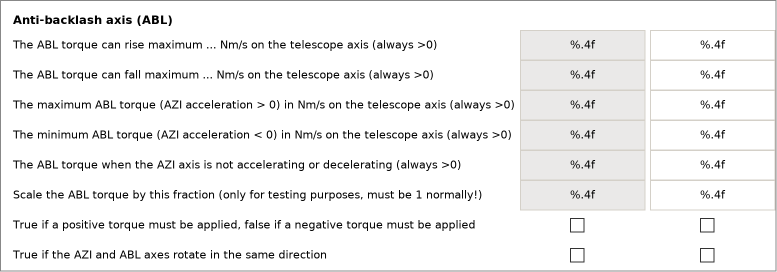
VISUALIZATION VISU_AxesConfig_Azimuth_3  // 777x272
VAR_IN_OUT
    active : AxesAzimuthConfig;
    editable : AxesAzimuthConfig;
END_VAR
    Label (10,5 205x30), "Anti-backlash axis (ABL)"
    Label (10,30 475x30), "The ABL torque can rise maximum ... Nm/s on the telescope axis (always >0)"
    Frame (520,30 255x30)
        shows VISU_ConfigLREAL4Entry(active := active.ablMaxTorqueRiseSpeed, editable := editable.ablMaxTorqueRiseSpeed)
    Label (10,60 475x30), "The ABL torque can fall maximum ... Nm/s on the telescope axis (always >0)"
    Label (10,90 505x30), "The maximum ABL torque (AZI acceleration > 0) in Nm/s on the telescope axis (always >0)"
    Label (10,120 500x30), "The minimum ABL torque (AZI acceleration < 0) in Nm/s on the telescope axis (always >0)"
    Label (10,150 500x30), "The ABL torque when the AZI axis is not accelerating or decelerating (always >0)"
    Label (10,180 500x30), "Scale the ABL torque by this fraction (only for testing purposes, must be 1 normally!)"
    Label (10,210 500x30), "True if a positive torque must be applied, false if a negative torque must be applied"
    Frame (520,210 255x30)
        shows VISU_ConfigBOOLEntry(active := active.ablPositiveTorque, editable := editable.ablPositiveTorque)
    Label (10,240 500x30), "True if the AZI and ABL axes rotate in the same direction"
    Frame (520,240 255x30)
        shows VISU_ConfigBOOLEntry(active := active.aziAndAblSameDirection, editable := editable.aziAndAblSameDirection)
    Frame (520,60 255x30)
        shows VISU_ConfigLREAL4Entry(active := active.ablMaxTorqueFallSpeed, editable := editable.ablMaxTorqueFallSpeed)
    Frame (520,90 255x30)
        shows VISU_ConfigLREAL4Entry(active := active.ablMaxTorque, editable := editable.ablMaxTorque)
    Frame (520,120 255x30)
        shows VISU_ConfigLREAL4Entry(active := active.ablMinTorque, editable := editable.ablMinTorque)
    Frame (520,150 255x30)
        shows VISU_ConfigLREAL4Entry(active := active.ablZeroAccTorque, editable := editable.ablZeroAccTorque)
    Frame (520,180 255x30)
        shows VISU_ConfigLREAL4Entry(active := active.ablTorqueOutputOverride, editable := editable.ablTorqueOutputOverride)
END_VISUALIZATION

// ---- MTCS/Axes/Visu/VISU_AxesConfig_Rotation_2.TcVIS
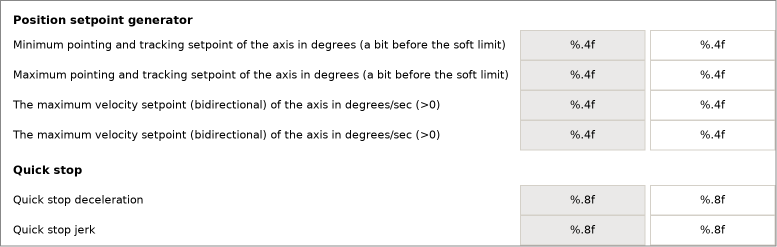
VISUALIZATION VISU_AxesConfig_Rotation_2  // 777x247
VAR_IN_OUT
    active : AxesRotationConfig;
    editable : AxesRotationConfig;
END_VAR
    Label (10,5 205x30), "Position setpoint generator"
    Label (10,30 495x30), "Minimum pointing and tracking setpoint of the axis in degrees (a bit before the soft limit)"
    Label (10,60 510x30), "Maximum pointing and tracking setpoint of the axis in degrees (a bit before the soft limit)"
    Label (10,90 475x30), "The maximum velocity setpoint (bidirectional) of the axis in degrees/sec (>0)"
    Label (10,120 475x30), "The maximum velocity setpoint (bidirectional) of the axis in degrees/sec (>0)"
    Frame (520,30 255x30)
        shows VISU_ConfigLREAL4Entry(active := active.minPositionSetpoint, editable := editable.minPositionSetpoint)
    Frame (520,60 255x30)
        shows VISU_ConfigLREAL4Entry(active := active.maxPositionSetpoint, editable := editable.maxPositionSetpoint)
    Frame (520,90 255x30)
        shows VISU_ConfigLREAL4Entry(active := active.maxVelocitySetpoint, editable := editable.maxVelocitySetpoint)
    Frame (520,120 255x30)
        shows VISU_ConfigLREAL4Entry(active := active.maxAccelerationSetpoint, editable := editable.maxAccelerationSetpoint)
    Label (10,155 205x30), "Quick stop"
    Frame (520,185 255x30)
        shows VISU_ConfigLREAL8Entry(active := active.quickStopDeceleration, editable := editable.quickStopDeceleration)
    Label (10,185 500x30), "Quick stop deceleration"
    Label (10,215 500x30), "Quick stop jerk"
    Frame (520,215 255x30)
        shows VISU_ConfigLREAL8Entry(active := active.quickStopJerk, editable := editable.quickStopJerk)
END_VISUALIZATION

// ---- MTCS/Axes/Visu/VISU_AxesConfig_Rotation_1.TcVIS
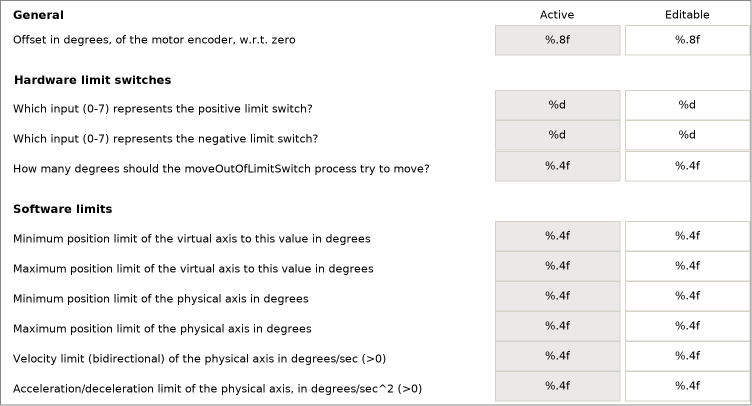
VISUALIZATION VISU_AxesConfig_Rotation_1  // 752x406
VAR_IN_OUT
    active : AxesRotationConfig;
    editable : AxesRotationConfig;
END_VAR
    Label (495,5 125x20), "Active"
    Label (625,5 125x20), "Editable"
    Label (10,25 360x30), "Offset in degrees, of the motor encoder, w.r.t. zero"
    Frame (495,25 255x30)
        shows VISU_ConfigLREAL8Entry(active := active.motorEncoderOffset, editable := editable.motorEncoderOffset)
    Label (10,94 475x30), "Which input (0-7) represents the positive limit switch?"
    Label (10,124 475x30), "Which input (0-7) represents the negative limit switch?"
    Label (10,154 475x30), "How many degrees should the moveOutOfLimitSwitch process try to move?"
    Label (11,65 150x30), "Hardware limit switches"
    Label (10,224 475x30), "Minimum position limit of the virtual axis to this value in degrees"
    Label (10,194 165x30), "Software limits"
    Label (10,254 475x30), "Maximum position limit of the virtual axis to this value in degrees"
    Label (10,284 475x30), "Minimum position limit of the physical axis in degrees"
    Label (10,314 475x30), "Maximum position limit of the physical axis in degrees"
    Label (10,344 475x30), "Velocity limit (bidirectional) of the physical axis in degrees/sec (>0)"
    Label (10,374 475x30), "Acceleration/deceleration limit of the physical axis, in degrees/sec^2 (>0)"
    Label (10,0 150x30), "General"
    Frame (495,90 255x30)
        shows VISU_ConfigSINTEntry(active := active.positiveLimitSwitchInput, editable := editable.positiveLimitSwitchInput)
    Frame (495,120 255x30)
        shows VISU_ConfigSINTEntry(active := active.negativeLimitSwitchInput, editable := editable.negativeLimitSwitchInput)
    Frame (495,151 255x30)
        shows VISU_ConfigLREAL4Entry(active := active.moveOutOfLimitSwitchDistance, editable := editable.moveOutOfLimitSwitchDistance)
    Frame (495,221 255x30)
        shows VISU_ConfigLREAL4Entry(active := active.minPositionLimitVirtualAxis, editable := editable.minPositionLimitVirtualAxis)
    Frame (495,251 255x30)
        shows VISU_ConfigLREAL4Entry(active := active.maxPositionLimitVirtualAxis, editable := editable.maxPositionLimitVirtualAxis)
    Frame (495,281 255x30)
        shows VISU_ConfigLREAL4Entry(active := active.minPositionLimitPhysicalAxis, editable := editable.minPositionLimitPhysicalAxis)
    Frame (495,311 255x30)
        shows VISU_ConfigLREAL4Entry(active := active.maxPositionLimitPhysicalAxis, editable := editable.maxPositionLimitPhysicalAxis)
    Frame (495,341 255x30)
        shows VISU_ConfigLREAL4Entry(active := active.velocityLimit, editable := editable.velocityLimit)
    Frame (495,371 255x30)
        shows VISU_ConfigLREAL4Entry(active := active.accelerationLimit, editable := editable.accelerationLimit)
END_VISUALIZATION

// ---- MTCS/Axes/Visu/VISU_AxesConfig_Elevation_2.TcVIS
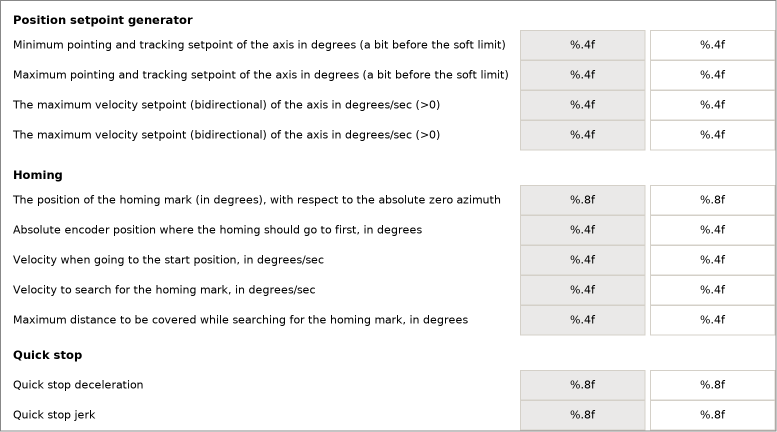
VISUALIZATION VISU_AxesConfig_Elevation_2  // 777x432
VAR_IN_OUT
    active : AxesElevationConfig;
    editable : AxesElevationConfig;
END_VAR
    Frame (520,185 255x30)
        shows VISU_ConfigLREAL8Entry(active := active.homingHomePosition, editable := editable.homingHomePosition)
    Label (10,185 500x30), "The position of the homing mark (in degrees), with respect to the absolute zero azimuth"
    Label (10,5 205x30), "Position setpoint generator"
    Label (10,30 490x30), "Minimum pointing and tracking setpoint of the axis in degrees (a bit before the soft limit)"
    Label (10,60 500x30), "Maximum pointing and tracking setpoint of the axis in degrees (a bit before the soft limit)"
    Label (10,90 475x30), "The maximum velocity setpoint (bidirectional) of the axis in degrees/sec (>0)"
    Label (10,120 475x30), "The maximum velocity setpoint (bidirectional) of the axis in degrees/sec (>0)"
    Label (10,160 205x30), "Homing"
    Label (10,215 475x30), "Absolute encoder position where the homing should go to first, in degrees"
    Label (10,245 475x30), "Velocity when going to the start position, in degrees/sec"
    Label (10,275 505x30), "Velocity to search for the homing mark, in degrees/sec"
    Label (10,305 500x30), "Maximum distance to be covered while searching for the homing mark, in degrees"
    Frame (520,30 255x30)
        shows VISU_ConfigLREAL4Entry(active := active.minPositionSetpoint, editable := editable.minPositionSetpoint)
    Frame (520,60 255x30)
        shows VISU_ConfigLREAL4Entry(active := active.maxPositionSetpoint, editable := editable.maxPositionSetpoint)
    Frame (520,90 255x30)
        shows VISU_ConfigLREAL4Entry(active := active.maxVelocitySetpoint, editable := editable.maxVelocitySetpoint)
    Frame (520,120 255x30)
        shows VISU_ConfigLREAL4Entry(active := active.maxAccelerationSetpoint, editable := editable.maxAccelerationSetpoint)
    Frame (520,215 255x30)
        shows VISU_ConfigLREAL4Entry(active := active.homingStartAbsEncPosition, editable := editable.homingStartAbsEncPosition)
    Frame (520,245 255x30)
        shows VISU_ConfigLREAL4Entry(active := active.homingGotoStartVelocity, editable := editable.homingGotoStartVelocity)
    Frame (520,275 255x30)
        shows VISU_ConfigLREAL4Entry(active := active.homingVelocity, editable := editable.homingVelocity)
    Frame (520,305 255x30)
        shows VISU_ConfigLREAL4Entry(active := active.homingRange, editable := editable.homingRange)
    Label (10,340 205x30), "Quick stop"
    Frame (520,370 255x30)
        shows VISU_ConfigLREAL8Entry(active := active.quickStopDeceleration, editable := editable.quickStopDeceleration)
    Label (10,370 500x30), "Quick stop deceleration"
    Label (10,400 500x30), "Quick stop jerk"
    Frame (520,400 255x30)
        shows VISU_ConfigLREAL8Entry(active := active.quickStopJerk, editable := editable.quickStopJerk)
END_VISUALIZATION

// ---- MTCS/Axes/Visu/VISU_AxesConfig_Elevation_1.TcVIS
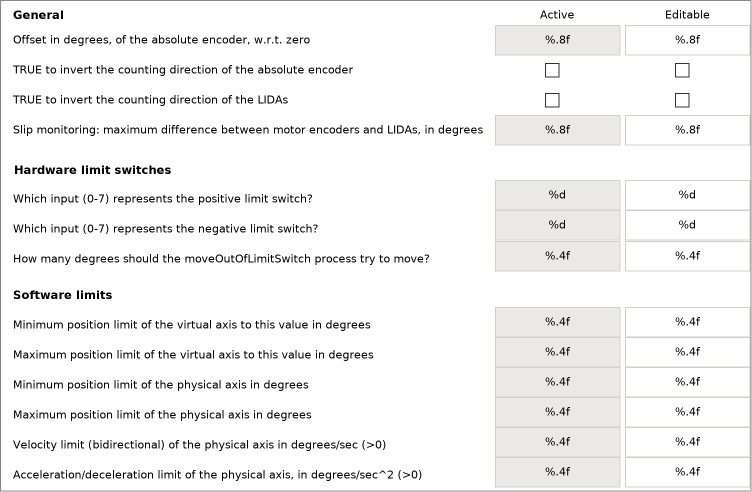
VISUALIZATION VISU_AxesConfig_Elevation_1  // 752x492
VAR_IN_OUT
    active : AxesElevationConfig;
    editable : AxesElevationConfig;
END_VAR
    Label (495,5 125x20), "Active"
    Label (625,5 125x20), "Editable"
    Label (10,25 360x30), "Offset in degrees, of the absolute encoder, w.r.t. zero"
    Frame (495,25 255x30)
        shows VISU_ConfigLREAL8Entry(active := active.absoluteEncoderOffset, editable := editable.absoluteEncoderOffset)
    Label (10,184 475x30), "Which input (0-7) represents the positive limit switch?"
    Label (10,214 475x30), "Which input (0-7) represents the negative limit switch?"
    Label (10,244 475x30), "How many degrees should the moveOutOfLimitSwitch process try to move?"
    Label (11,155 150x30), "Hardware limit switches"
    Label (10,310 475x30), "Minimum position limit of the virtual axis to this value in degrees"
    Label (10,280 165x30), "Software limits"
    Label (10,340 475x30), "Maximum position limit of the virtual axis to this value in degrees"
    Label (10,370 475x30), "Minimum position limit of the physical axis in degrees"
    Label (10,400 475x30), "Maximum position limit of the physical axis in degrees"
    Label (10,430 475x30), "Velocity limit (bidirectional) of the physical axis in degrees/sec (>0)"
    Label (10,460 475x30), "Acceleration/deceleration limit of the physical axis, in degrees/sec^2 (>0)"
    Label (10,115 480x30), "Slip monitoring: maximum difference between motor encoders and LIDAs, in degrees"
    Frame (495,115 255x30)
        shows VISU_ConfigLREAL8Entry(active := active.slipLimit, editable := editable.slipLimit)
    Label (10,0 150x30), "General"
    Frame (495,180 255x30)
        shows VISU_ConfigSINTEntry(active := active.positiveLimitSwitchInput, editable := editable.positiveLimitSwitchInput)
    Frame (495,210 255x30)
        shows VISU_ConfigSINTEntry(active := active.negativeLimitSwitchInput, editable := editable.negativeLimitSwitchInput)
    Frame (495,241 255x30)
        shows VISU_ConfigLREAL4Entry(active := active.moveOutOfLimitSwitchDistance, editable := editable.moveOutOfLimitSwitchDistance)
    Frame (495,307 255x30)
        shows VISU_ConfigLREAL4Entry(active := active.minPositionLimitVirtualAxis, editable := editable.minPositionLimitVirtualAxis)
    Frame (495,337 255x30)
        shows VISU_ConfigLREAL4Entry(active := active.maxPositionLimitVirtualAxis, editable := editable.maxPositionLimitVirtualAxis)
    Frame (495,367 255x30)
        shows VISU_ConfigLREAL4Entry(active := active.minPositionLimitPhysicalAxis, editable := editable.minPositionLimitPhysicalAxis)
    Frame (495,397 255x30)
        shows VISU_ConfigLREAL4Entry(active := active.maxPositionLimitPhysicalAxis, editable := editable.maxPositionLimitPhysicalAxis)
    Frame (495,427 255x30)
        shows VISU_ConfigLREAL4Entry(active := active.velocityLimit, editable := editable.velocityLimit)
    Frame (495,457 255x30)
        shows VISU_ConfigLREAL4Entry(active := active.accelerationLimit, editable := editable.accelerationLimit)
    Frame (495,55 255x30)
        shows VISU_ConfigBOOLEntry(active := active.absoluteEncoderInvert, editable := editable.absoluteEncoderInvert)
    Label (10,55 360x30), "TRUE to invert the counting direction of the absolute encoder"
    Frame (495,85 255x30)
        shows VISU_ConfigBOOLEntry(active := active.lidasInvert, editable := editable.lidasInvert)
    Label (10,85 360x30), "TRUE to invert the counting direction of the LIDAs"
END_VISUALIZATION

// ---- MTCS/Axes/Visu/VISU_AxesConfig_Azimuth_2.TcVIS
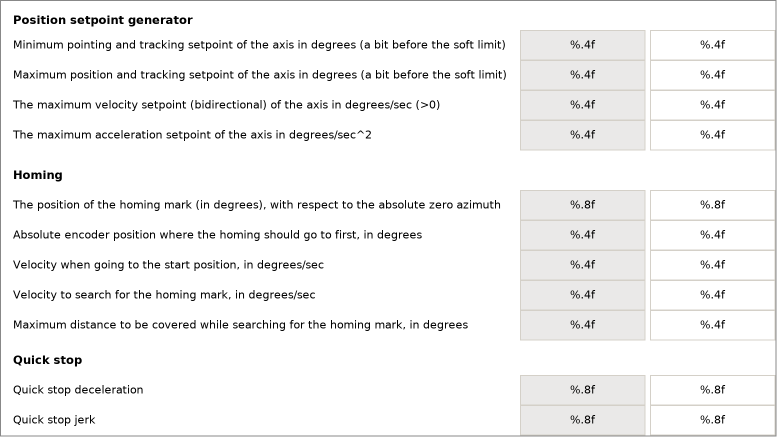
VISUALIZATION VISU_AxesConfig_Azimuth_2  // 777x437
VAR_IN_OUT
    active : AxesAzimuthConfig;
    editable : AxesAzimuthConfig;
END_VAR
    Frame (520,190 255x30)
        shows VISU_ConfigLREAL8Entry(active := active.homingHomePosition, editable := editable.homingHomePosition)
    Label (10,5 205x30), "Position setpoint generator"
    Label (10,30 500x30), "Minimum pointing and tracking setpoint of the axis in degrees (a bit before the soft limit)"
    Frame (520,30 255x30)
        shows VISU_ConfigLREAL4Entry(active := active.minPositionSetpoint, editable := editable.minPositionSetpoint)
    Label (10,60 500x30), "Maximum position and tracking setpoint of the axis in degrees (a bit before the soft limit)"
    Label (10,90 475x30), "The maximum velocity setpoint (bidirectional) of the axis in degrees/sec (>0)"
    Label (10,120 475x30), "The maximum acceleration setpoint of the axis in degrees/sec^2"
    Label (10,160 205x30), "Homing"
    Label (10,220 475x30), "Absolute encoder position where the homing should go to first, in degrees"
    Label (10,250 475x30), "Velocity when going to the start position, in degrees/sec"
    Label (10,280 505x30), "Velocity to search for the homing mark, in degrees/sec"
    Label (10,310 500x30), "Maximum distance to be covered while searching for the homing mark, in degrees"
    Frame (520,60 255x30)
        shows VISU_ConfigLREAL4Entry(active := active.maxPositionSetpoint, editable := editable.maxPositionSetpoint)
    Frame (520,90 255x30)
        shows VISU_ConfigLREAL4Entry(active := active.maxVelocitySetpoint, editable := editable.maxVelocitySetpoint)
    Frame (520,120 255x30)
        shows VISU_ConfigLREAL4Entry(active := active.maxAccelerationSetpoint, editable := editable.maxAccelerationSetpoint)
    Frame (520,220 255x30)
        shows VISU_ConfigLREAL4Entry(active := active.homingStartAbsEncPosition, editable := editable.homingStartAbsEncPosition)
    Frame (520,250 255x30)
        shows VISU_ConfigLREAL4Entry(active := active.homingGotoStartVelocity, editable := editable.homingGotoStartVelocity)
    Frame (520,280 255x30)
        shows VISU_ConfigLREAL4Entry(active := active.homingVelocity, editable := editable.homingVelocity)
    Frame (520,310 255x30)
        shows VISU_ConfigLREAL4Entry(active := active.homingRange, editable := editable.homingRange)
    Label (10,190 500x30), "The position of the homing mark (in degrees), with respect to the absolute zero azimuth"
    Label (10,345 205x30), "Quick stop"
    Frame (520,375 255x30)
        shows VISU_ConfigLREAL8Entry(active := active.quickStopDeceleration, editable := editable.quickStopDeceleration)
    Label (10,375 500x30), "Quick stop deceleration"
    Label (10,405 500x30), "Quick stop jerk"
    Frame (520,405 255x30)
        shows VISU_ConfigLREAL8Entry(active := active.quickStopJerk, editable := editable.quickStopJerk)
END_VISUALIZATION

// ---- MTCS/Axes/Visu/VISU_AxesConfig_FilterWheel.TcVIS
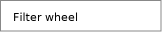
VISUALIZATION VISU_AxesConfig_FilterWheel  // 162x32
    Label (10,5 150x25), "Filter wheel"
END_VISUALIZATION

// ---- MTCS/Axes/Visu/VISU_AxesElevationAxis.TcVIS
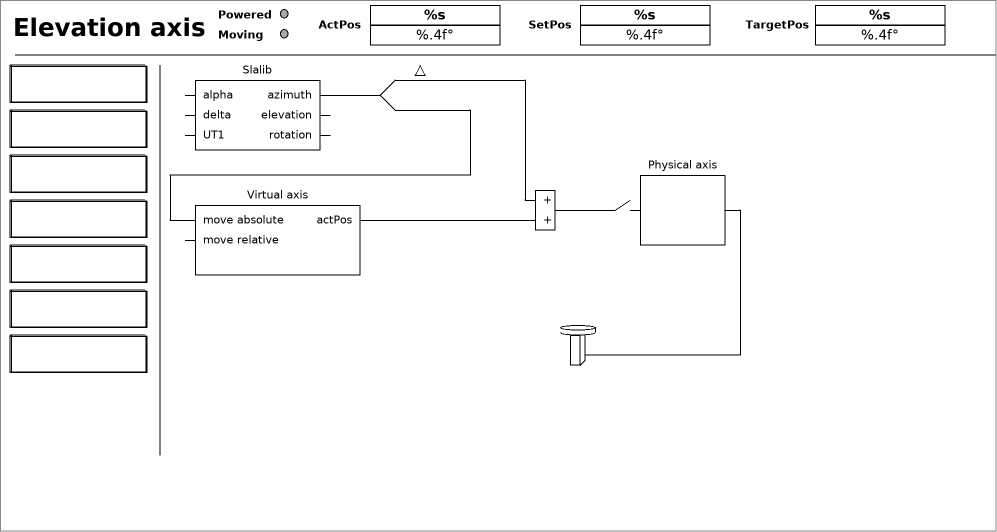
VISUALIZATION VISU_AxesElevationAxis  // 997x532
VAR_IN_OUT
	ref : AxesElevationAxis;
    ref_driveChannel : AX52XXDriveChannel;
    widget : AxesElevationAxisWidget;
END_VAR
    Rectangle (10,5 590x45), "Elevation axis"
    Frame (10,65 140x40)
        shows VISU_SubSubSystemButton(widget := widget.button_overview)
        OnMouseClick: FrameSelectionChange Selection=SelectedFrame=e720f99c-78fc-49d3-920d-5c22fdf0231f, GlobSel=AssignType=Directly, SelType=Locally
        OnMouseClick: execute { widget.activeTab := AxesElevationAxisTabs.OVERVIEW; }
    Frame (165,60 805x470)
        shows VISU_AxesElevationAxis_Overview(ref := ref, widget := widget)
        shows VISU_AxesElevationAxis_Processes(ref := ref, ref_driveChannel := ref_driveChannel, widget := widget)
        shows VISU_AX522DriveChannel(ref := ref_driveChannel, widget := widget.driveChannel)
        shows VISU_AngularAxis(axis := ref.parts.virtualAxis, widget := widget.virtualAxis)
        shows VISU_AngularAxis(axis := ref.parts.physicalAxis, widget := widget.physicalAxis)
        shows VISU_AxesElevationAxis_Lidas(ref := ref, widget := widget)
        shows VISU_AxesElevationAxis_AbsoluteEncoder(ref := ref, widget := widget)
        shows VISU_AxesAzimuthAxis_AbsoluteEncoder(ref := ref, widget := widget)
        p3523098516: ref
    Line (160,455) (160,65)
    Frame (10,155 140x40)
        shows VISU_SubSubSystemButton(widget := widget.button_driveChannel)
        OnMouseClick: FrameSelectionChange Selection=SelectedFrame=e720f99c-78fc-49d3-920d-5c22fdf0231f, Selection=2, GlobSel=AssignType=Directly, SelType=Locally
        OnMouseClick: execute { widget.activeTab := AxesElevationAxisTabs.DRIVE_CHANNEL; }
    Frame (10,200 140x40)
        shows VISU_SubSubSystemButton(widget := widget.button_virtualAxis)
        OnMouseClick: FrameSelectionChange Selection=SelectedFrame=e720f99c-78fc-49d3-920d-5c22fdf0231f, Selection=3, GlobSel=AssignType=Directly, SelType=Locally
        OnMouseClick: execute { widget.activeTab := AxesElevationAxisTabs.VIRTUAL_AXIS; }
    Frame (10,245 140x40)
        shows VISU_SubSubSystemButton(widget := widget.button_physicalAxis)
        OnMouseClick: FrameSelectionChange Selection=SelectedFrame=e720f99c-78fc-49d3-920d-5c22fdf0231f, Selection=4, GlobSel=AssignType=Directly, SelType=Locally
        OnMouseClick: execute { widget.activeTab := AxesElevationAxisTabs.PHYSICAL_AXIS; }
    Frame (10,290 140x40)
        shows VISU_SubSubSystemButton(widget := widget.button_lidas)
        OnMouseClick: FrameSelectionChange Selection=SelectedFrame=e720f99c-78fc-49d3-920d-5c22fdf0231f, Selection=5, GlobSel=AssignType=Directly, SelType=Locally
        OnMouseClick: execute { widget.activeTab := AxesElevationAxisTabs.LIDAS; }
    Frame (10,335 140x40)
        shows VISU_SubSubSystemButton(widget := widget.button_absoluteEncoder)
        OnMouseClick: FrameSelectionChange Selection=SelectedFrame=e720f99c-78fc-49d3-920d-5c22fdf0231f, Selection=6, GlobSel=AssignType=Directly, SelType=Locally
        OnMouseClick: execute { widget.activeTab := AxesElevationAxisTabs.ABSOLUTE_ENCODER; }
    Frame (10,110 140x40)
        shows VISU_SubSubSystemButton(widget := widget.button_processes)
        OnMouseClick: FrameSelectionChange Selection=SelectedFrame=e720f99c-78fc-49d3-920d-5c22fdf0231f, Selection=1, GlobSel=AssignType=Directly, SelType=Locally
        OnMouseClick: execute { widget.activeTab := AxesElevationAxisTabs.PROCESSES; }
    Line (995,55) (15,55)
    Label (310,0 60x50), "ActPos"
    Rectangle (370,5 130x20), "%s", text variable: widget.actPos.dmsString
    Rectangle (370,25 130x20), "%.4f°", text variable: ref.actPos.degrees.value
    Label (520,0 60x50), "SetPos"
    Rectangle (580,5 130x20), "%s", text variable: widget.setPos.dmsString
    Rectangle (580,25 130x20), "%.4f°", text variable: ref.setPos.degrees.value
    Label (740,0 75x50), "TargetPos"
    Rectangle (815,5 130x20), "%s", text variable: widget.targetPos.dmsString
    Rectangle (815,25 130x20), "%.4f°", text variable: ref.targetPos.degrees.value
    Label (215,5 65x20), "Powered"
    Frame (280,5 10x15)
        shows VISU_State_gray_green(state := ref.statuses.poweredStatus.enabled)
    Label (215,25 65x20), "Moving"
    Frame (280,25 10x15)
        shows VISU_State_gray_green(state := ref.parts.physicalAxis.axis_ref.Status.Moving)
END_VISUALIZATION

// ---- MTCS/Axes/Visu/VISU_AxesExternalSetpointGenerator.TcVIS
VISUALIZATION VISU_AxesExternalSetpointGenerator  // 2x2
END_VISUALIZATION

// ---- MTCS/Axes/Visu/VISU_AxesRotationAxis.TcVIS
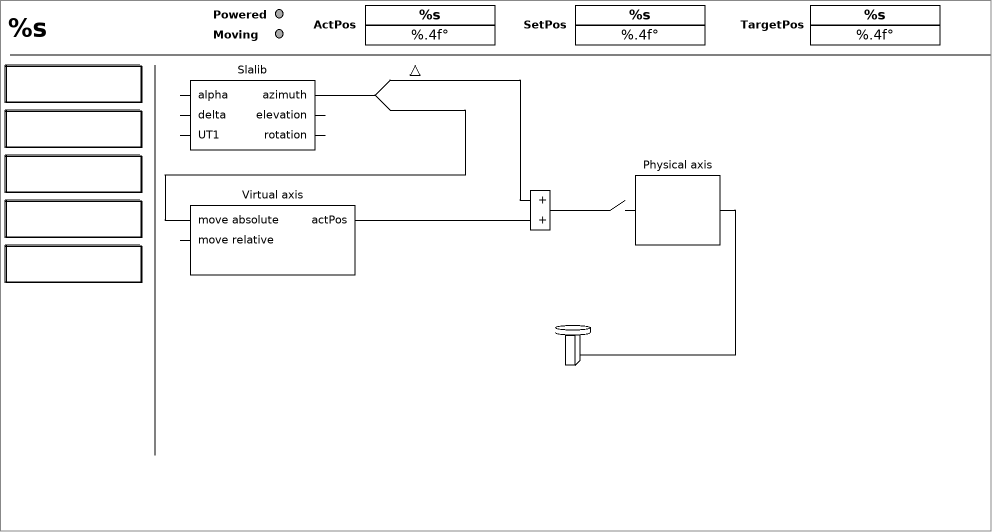
VISUALIZATION VISU_AxesRotationAxis  // 992x532
VAR_IN_OUT
	ref : AxesRotationAxis;
    ref_driveChannel : AX52XXDriveChannel;
    widget : AxesRotationAxisWidget;
END_VAR
    Frame (5,65 140x40)
        shows VISU_SubSubSystemButton(widget := widget.button_overview)
        OnMouseClick: FrameSelectionChange Selection=SelectedFrame=b6fa029b-3640-42a1-bfcc-db8ab31a5104, GlobSel=AssignType=Directly, SelType=Locally
        OnMouseClick: execute { widget.activeTab := AxesRotationAxisTabs.OVERVIEW; }
    Frame (160,60 805x470)
        shows VISU_AxesRotationAxis_Overview(ref := ref, widget := widget)
        shows VISU_AxesRotationAxis_Processes(ref := ref, ref_driveChannel := ref_driveChannel, widget := widget)
        shows VISU_AX522DriveChannel(ref := ref_driveChannel, widget := widget.driveChannel)
        shows VISU_AngularAxis(axis := ref.parts.virtualAxis, widget := widget.virtualAxis)
        shows VISU_AngularAxis(axis := ref.parts.physicalAxis, widget := widget.physicalAxis)
        shows VISU_AxesElevationAxis_AbsoluteEncoder(ref := ref, widget := widget)
        shows VISU_AxesAzimuthAxis_AbsoluteEncoder(ref := ref, widget := widget)
        shows VISU_AxesElevationAxis_Lidas(ref := ref, widget := widget)
        p3523098516: ref
    Line (155,455) (155,65)
    Frame (5,155 140x40)
        shows VISU_SubSubSystemButton(widget := widget.button_driveChannel)
        OnMouseClick: FrameSelectionChange Selection=SelectedFrame=b6fa029b-3640-42a1-bfcc-db8ab31a5104, Selection=2, GlobSel=AssignType=Directly, SelType=Locally
        OnMouseClick: execute { widget.activeTab := AxesRotationAxisTabs.DRIVE_CHANNEL; }
    Frame (5,200 140x40)
        shows VISU_SubSubSystemButton(widget := widget.button_virtualAxis)
        OnMouseClick: FrameSelectionChange Selection=SelectedFrame=b6fa029b-3640-42a1-bfcc-db8ab31a5104, Selection=3, GlobSel=AssignType=Directly, SelType=Locally
        OnMouseClick: execute { widget.activeTab := AxesRotationAxisTabs.VIRTUAL_AXIS; }
    Frame (5,245 140x40)
        shows VISU_SubSubSystemButton(widget := widget.button_physicalAxis)
        OnMouseClick: FrameSelectionChange Selection=SelectedFrame=b6fa029b-3640-42a1-bfcc-db8ab31a5104, Selection=4, GlobSel=AssignType=Directly, SelType=Locally
        OnMouseClick: execute { widget.activeTab := AxesRotationAxisTabs.PHYSICAL_AXIS; }
    Frame (5,110 140x40)
        shows VISU_SubSubSystemButton(widget := widget.button_processes)
        OnMouseClick: FrameSelectionChange Selection=SelectedFrame=b6fa029b-3640-42a1-bfcc-db8ab31a5104, Selection=1, GlobSel=AssignType=Directly, SelType=Locally
        OnMouseClick: execute { widget.activeTab := AxesRotationAxisTabs.PROCESSES; }
    Line (990,55) (10,55)
    Label (305,0 60x50), "ActPos"
    Rectangle (365,5 130x20), "%s", text variable: widget.actPos.dmsString
    Rectangle (365,25 130x20), "%.4f°", text variable: ref.actPos.degrees.value
    Label (515,0 60x50), "SetPos"
    Rectangle (575,5 130x20), "%s", text variable: widget.setPos.dmsString
    Rectangle (575,25 130x20), "%.4f°", text variable: ref.setPos.degrees.value
    Label (735,0 75x50), "TargetPos"
    Rectangle (810,5 130x20), "%s", text variable: widget.targetPos.dmsString
    Rectangle (810,25 130x20), "%.4f°", text variable: ref.targetPos.degrees.value
    Label (210,5 65x20), "Powered"
    Frame (275,5 10x15)
        shows VISU_State_gray_green(state := ref.statuses.poweredStatus.enabled)
    Label (210,25 65x20), "Moving"
    Frame (275,25 10x15)
        shows VISU_State_gray_green(state := ref.parts.physicalAxis.axis_ref.Status.Moving)
    Rectangle (5,5 200x46), "%s", text variable: widget.axisTitle
END_VISUALIZATION

// ---- MTCS/Axes/Visu/VISU_AxesManual.TcVIS
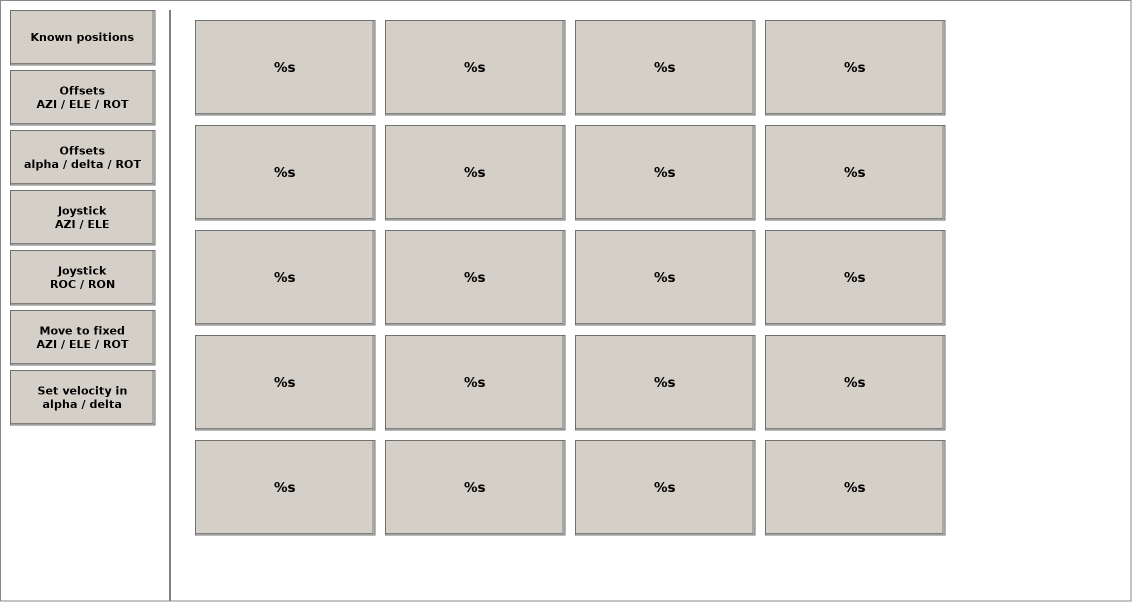
VISUALIZATION VISU_AxesManual  // 1132x602
VAR_IN_OUT
	ref : Axes;
    widget : AxesManualWidget;
END_VAR
    Button (10,10 145x55), "Known positions", pressed state: widget.activeTab = AxesManualTabs.TAB_POSITIONS
        OnMouseClick: execute { widget.activeTab := AxesManualTabs.TAB_POSITIONS; }
    Button (10,190 145x55), "Joystick AZI / ELE", pressed state: widget.activeTab = AxesManualTabs.TAB_JOYSTICK_AZIELE
        OnMouseClick: execute { widget.activeTab := AxesManualTabs.TAB_JOYSTICK_AZIELE; }
    Button (10,250 145x55), "Joystick ROC / RON", pressed state: widget.activeTab = AxesManualTabs.TAB_JOYSTICK_ROT
        OnMouseClick: execute { widget.activeTab := AxesManualTabs.TAB_JOYSTICK_ROT; }
    Button (10,70 145x55), "Offsets AZI / ELE / ROT", pressed state: widget.activeTab = AxesManualTabs.TAB_OFFSETS_AZIELE
        OnMouseClick: execute { widget.activeTab := AxesManualTabs.TAB_OFFSETS_AZIELE; }
    Button (10,310 145x55), "Move to fixed AZI / ELE / ROT", pressed state: widget.activeTab = AxesManualTabs.TAB_MOVEABSOLUTE
        OnMouseClick: execute { widget.activeTab := AxesManualTabs.TAB_MOVEABSOLUTE; }
    Button (10,370 145x55), "Set velocity in alpha / delta", pressed state: widget.activeTab = AxesManualTabs.TAB_MOVEVELOCITY
        OnMouseClick: execute { widget.activeTab := AxesManualTabs.TAB_MOVEVELOCITY; }
    Line (170,600) (170,10)
    Frame (180,10 950x590), frame switch variable: widget.activeTab
        shows VISU_AxesManual_Positions(ref := ref, widget := widget.positions)
        shows VISU_AxesManual_Joystick_AziEle(ref := ref, widget := widget.joystickAziEle)
        shows VISU_AxesManual_Joystick_Rot(ref := ref, widget := widget.joystickRot)
        shows VISU_AxesManual_Offsets_AziEleRot(ref := ref, widget := widget.offsets)
        shows VISU_AxesManual_Offsets_AlphaDeltaRot(ref := ref, widget := widget.offsets)
        shows VISU_AxesManual_MoveAbsolute(ref := ref, widget := widget.moveAbsolute)
        shows VISU_AxesManual_MoveVelocity(ref := ref, widget := widget.moveVelocity)
    Button (10,130 145x55), "Offsets alpha / delta / ROT", pressed state: widget.activeTab = AxesManualTabs.TAB_OFFSETS_ALPHADELTA
        OnMouseClick: execute { widget.activeTab := AxesManualTabs.TAB_OFFSETS_ALPHADELTA; }
END_VISUALIZATION

// ---- MTCS/Axes/Visu/VISU_AxesConfig.TcVIS
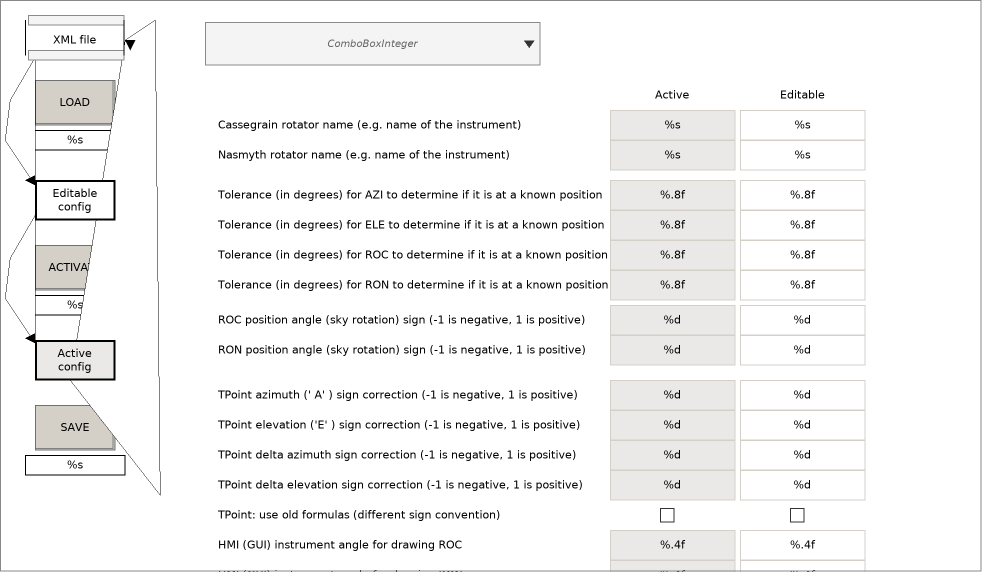
VISUALIZATION VISU_AxesConfig  // 982x572
VAR_IN_OUT
    editable : AxesConfig;
	active : AxesConfig;
    mgr : ConfigManager;
    mgrWidget : ConfigManagerWidget;
    axesWidget : AxesWidget;
END_VAR
    Frame (10,5 180x495)
        shows VISU_ConfigManager(mgr := mgr, widget := mgrWidget)
    ComboBoxInteger (205,22 335x43), variable: axesWidget.activeConfigTab, text list: 'AxesConfigTextList'
    Frame (205,85 775x485), frame switch variable: axesWidget.activeConfigTab
        shows VISU_AxesConfig_General(editable := editable, active := active)
        shows VISU_AxesConfig_KnownPositions(activePosition := axesWidget.activeConfigPosition, editable := editable.knownPositions, active := active.knownPositions)
        shows VISU_AxesConfig_Location(active := active.location, editable := editable.location)
        shows VISU_AxesConfig_LocalConditions(active := active.localConditions, editable := editable.localConditions)
        shows VISU_AxesConfig_Azimuth_1(active := active.azi, editable := editable.azi)
        shows VISU_AxesConfig_Azimuth_2(active := active.azi, editable := editable.azi)
        shows VISU_AxesConfig_Azimuth_3(active := active.azi, editable := editable.azi)
        shows VISU_AxesConfig_Elevation_1(active := active.ele, editable := editable.ele)
        shows VISU_AxesConfig_Elevation_2(active := active.ele, editable := editable.ele)
        shows VISU_AxesConfig_Rotation_1(active := active.roc, editable := editable.roc)
        shows VISU_AxesConfig_Rotation_2(active := active.roc, editable := editable.roc)
        shows VISU_AxesConfig_Rotation_1(active := active.ron, editable := editable.ron)
        shows VISU_AxesConfig_Rotation_2(active := active.ron, editable := editable.ron)
        shows VISU_AxesConfig_FilterWheel()
        shows VISU_MeasurementConfig(active := active.relativeHumidities.insideTube, editable := editable.relativeHumidities.insideTube)
        shows VISU_MeasurementConfig(active := active.dewpoints.topAir, editable := editable.dewpoints.topAir)
        shows VISU_MeasurementConfig(active := active.dewpoints.insideTube, editable := editable.dewpoints.insideTube)
        shows VISU_MeasurementConfig(active := active.accelerometers.tube.x, editable := editable.accelerometers.tube.x)
        shows VISU_MeasurementConfig(active := active.accelerometers.tube.y, editable := editable.accelerometers.tube.y)
        p1226617324: active.relativeHumidities.topAir
        p1437654724: editable.relativeHumidities.topAir
END_VISUALIZATION

// ---- MTCS/Axes/Visu/VISU_AxesAxes.TcVIS
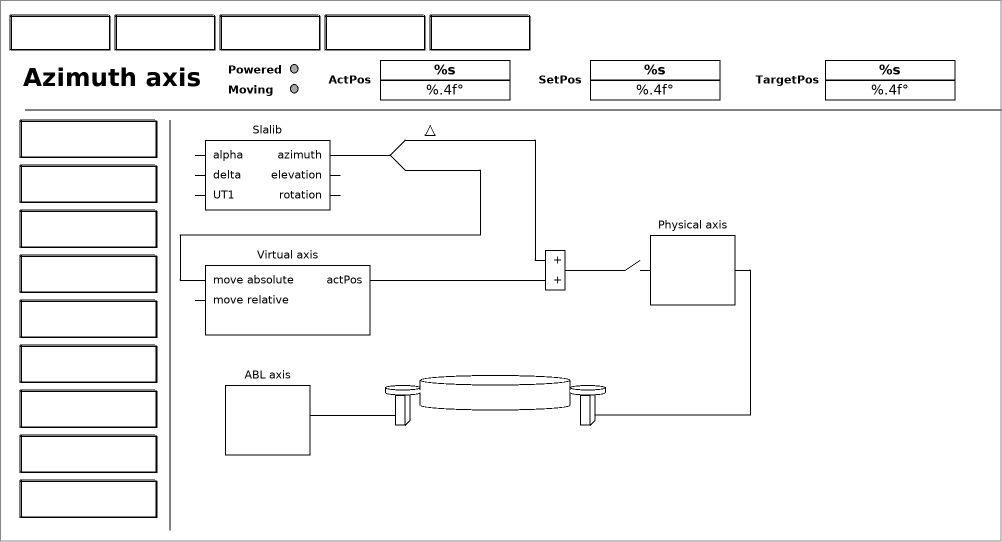
VISUALIZATION VISU_AxesAxes  // 1002x542
VAR_IN_OUT
    ref : Axes;
    widget : AxesAxesWidget;
END_VAR
    Frame (10,15 100x40)
        shows VISU_SubSubSystemButton(widget := widget.button_azi)
        OnMouseClick: FrameSelectionChange Selection=SelectedFrame=849b1b6c-774b-4476-bff7-38dbb17a175e, GlobSel=AssignType=Directly, SelType=Locally
        OnMouseClick: execute { widget.activeTab := AxesAxesTabs.AZI; }
    Frame (10,55 990x485)
        shows VISU_AxesAzimuthAxis(ref := ref.parts.azi, ref_aziDriveChannel := ref.parts.io.parts.aziDrive.parts.channelA, ref_ablDriveChannel := ref.parts.io.parts.ablDrive.parts.channelA, widget := widget.azi)
        shows VISU_AxesElevationAxis(ref := ref.parts.ele, ref_driveChannel := ref.parts.io.parts.eleDrive.parts.channelA, widget := widget.ele)
        shows VISU_AxesRotationAxis(ref := ref.parts.roc, ref_driveChannel := ref.parts.io.parts.aziDrive.parts.channelB, widget := widget.roc)
        shows VISU_AxesRotationAxis(ref := ref.parts.ron, ref_driveChannel := ref.parts.io.parts.ablDrive.parts.channelB, widget := widget.ron)
    Frame (115,15 100x40)
        shows VISU_SubSubSystemButton(widget := widget.button_ele)
        OnMouseClick: FrameSelectionChange Selection=SelectedFrame=849b1b6c-774b-4476-bff7-38dbb17a175e, Selection=1, GlobSel=AssignType=Directly, SelType=Locally
        OnMouseClick: execute { widget.activeTab := AxesAxesTabs.ELE; }
    Frame (220,15 100x40)
        shows VISU_SubSubSystemButton(widget := widget.button_roc)
        OnMouseClick: FrameSelectionChange Selection=SelectedFrame=849b1b6c-774b-4476-bff7-38dbb17a175e, Selection=2, GlobSel=AssignType=Directly, SelType=Locally
        OnMouseClick: execute { widget.activeTab := AxesAxesTabs.ROC; }
    Frame (325,15 100x40)
        shows VISU_SubSubSystemButton(widget := widget.button_ron)
        OnMouseClick: FrameSelectionChange Selection=SelectedFrame=849b1b6c-774b-4476-bff7-38dbb17a175e, Selection=3, GlobSel=AssignType=Directly, SelType=Locally
        OnMouseClick: execute { widget.activeTab := AxesAxesTabs.RON; }
    Frame (430,15 100x40)
        shows VISU_SubSubSystemButton(widget := widget.button_fw)
        OnMouseClick: FrameSelectionChange Selection=SelectedFrame=849b1b6c-774b-4476-bff7-38dbb17a175e, GlobSel=AssignType=Directly, SelType=Locally
        OnMouseClick: execute { widget.activeTab := AxesAxesTabs.FW; }
END_VISUALIZATION

// ---- MTCS/Axes/Visu/VISU_AxesAdvanced.TcVIS
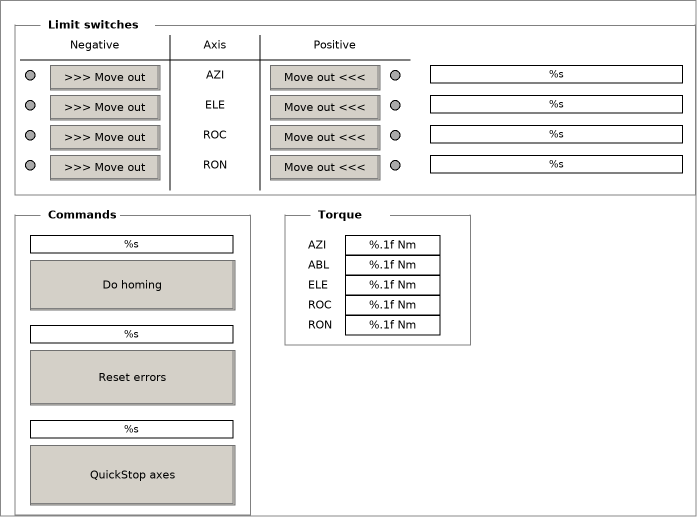
VISUALIZATION VISU_AxesAdvanced  // 697x517
VAR_IN_OUT
	ref : Axes;
    widget : AxesWidget;
END_VAR
    Polyline (120,215) (250,215) (250,515) (15,515) (15,215) (40,215)
    Polyline (155,25) (695,25) (695,195) (15,195) (15,25) (40,25)
    Label (45,15 100x20), "Limit switches"
    Label (170,60 90x30), "AZI"
    Frame (390,65 20x20)
        shows VISU_State_gray_red(state := ref.parts.azi.positiveLimitSwitchError)
    Line (260,190) (260,35)
    Line (170,190) (170,35)
    Label (260,30 150x30), "Positive"
    Label (20,30 150x30), "Negative"
    Line (410,60) (20,60)
    Label (170,30 90x30), "Axis"
    Button (270,65 110x25), "Move out <<<", input disabled if: ref.parts.azi.processes.moveOutOfLimitSwitch.statuses.enabledStatus.disabled
        OnMouseClick: execute { ref.parts.azi.processes.moveOutOfLimitSwitch.set.switch := LimitSwitches.POSITIVE_LIMIT_SWITCH; ref.parts.azi.processes.moveOutOfLimitSwitch.do_request := TRUE; }
    Frame (25,65 20x20)
        shows VISU_State_gray_red(state := ref.parts.azi.negativeLimitSwitchError)
    Button (50,65 110x25), ">>> Move out", input disabled if: ref.parts.azi.processes.moveOutOfLimitSwitch.statuses.enabledStatus.disabled
        OnMouseClick: execute { ref.parts.azi.processes.moveOutOfLimitSwitch.set.switch := LimitSwitches.NEGATIVE_LIMIT_SWITCH; ref.parts.azi.processes.moveOutOfLimitSwitch.do_request := TRUE; }
    Label (170,90 90x30), "ELE"
    Frame (390,95 20x20)
        shows VISU_State_gray_red(state := ref.parts.ele.positiveLimitSwitchError)
    Button (270,95 110x25), "Move out <<<", input disabled if: ref.parts.ele.processes.moveOutOfLimitSwitch.statuses.enabledStatus.disabled
        OnMouseClick: execute { ref.parts.ele.processes.moveOutOfLimitSwitch.set.switch := LimitSwitches.POSITIVE_LIMIT_SWITCH; ref.parts.ele.processes.moveOutOfLimitSwitch.do_request := TRUE; }
    Frame (25,95 20x20)
        shows VISU_State_gray_red(state := ref.parts.ele.negativeLimitSwitchError)
    Button (50,95 110x25), ">>> Move out", input disabled if: ref.parts.ele.processes.moveOutOfLimitSwitch.statuses.enabledStatus.disabled
        OnMouseClick: execute { ref.parts.ele.processes.moveOutOfLimitSwitch.set.switch := LimitSwitches.NEGATIVE_LIMIT_SWITCH; ref.parts.ele.processes.moveOutOfLimitSwitch.do_request := TRUE; }
    Label (170,120 90x30), "ROC"
    Frame (390,125 20x20)
        shows VISU_State_gray_red(state := ref.parts.roc.positiveLimitSwitchError)
    Button (270,125 110x25), "Move out <<<", input disabled if: ref.parts.roc.processes.moveOutOfLimitSwitch.statuses.enabledStatus.disabled
        OnMouseClick: execute { ref.parts.roc.processes.moveOutOfLimitSwitch.set.switch := LimitSwitches.POSITIVE_LIMIT_SWITCH; ref.parts.roc.processes.moveOutOfLimitSwitch.do_request := TRUE; }
    Frame (25,125 20x20)
        shows VISU_State_gray_red(state := ref.parts.roc.negativeLimitSwitchError)
    Button (50,125 110x25), ">>> Move out", input disabled if: ref.parts.roc.processes.moveOutOfLimitSwitch.statuses.enabledStatus.disabled
        OnMouseClick: execute { ref.parts.roc.processes.moveOutOfLimitSwitch.set.switch := LimitSwitches.NEGATIVE_LIMIT_SWITCH; ref.parts.roc.processes.moveOutOfLimitSwitch.do_request := TRUE; }
    Label (170,150 90x30), "RON"
    Frame (390,155 20x20)
        shows VISU_State_gray_red(state := ref.parts.ron.positiveLimitSwitchError)
    Button (270,155 110x25), "Move out <<<", input disabled if: ref.parts.ron.processes.moveOutOfLimitSwitch.statuses.enabledStatus.disabled
        OnMouseClick: execute { ref.parts.ron.processes.moveOutOfLimitSwitch.set.switch := LimitSwitches.POSITIVE_LIMIT_SWITCH; ref.parts.ron.processes.moveOutOfLimitSwitch.do_request := TRUE; }
    Frame (25,155 20x20)
        shows VISU_State_gray_red(state := ref.parts.ron.negativeLimitSwitchError)
    Button (50,155 110x25), ">>> Move out", input disabled if: ref.parts.ron.processes.moveOutOfLimitSwitch.statuses.enabledStatus.disabled
        OnMouseClick: execute { ref.parts.ron.processes.moveOutOfLimitSwitch.set.switch := LimitSwitches.NEGATIVE_LIMIT_SWITCH; ref.parts.ron.processes.moveOutOfLimitSwitch.do_request := TRUE; }
    Frame (430,65 255x20)
        shows VISU_StatusWidget(widget := widget.axes.azi.processes_moveOutOfLimitSwitchStatus)
    Frame (430,95 255x20)
        shows VISU_StatusWidget(widget := widget.axes.ele.processes_moveOutOfLimitSwitchStatus)
    Frame (430,125 255x20)
        shows VISU_StatusWidget(widget := widget.axes.roc.processes_moveOutOfLimitSwitchStatus)
    Frame (430,155 255x20)
        shows VISU_StatusWidget(widget := widget.axes.ron.processes_moveOutOfLimitSwitchStatus)
    Button (30,260 205x50), "Do homing", input disabled if: ref.processes.doHoming.statuses.enabledStatus.disabled
        OnMouseClick: execute { ref.processes.doHoming.do_request := TRUE; }
    Label (45,205 85x20), "Commands"
    Button (30,350 205x55), "Reset errors", input disabled if: ref.processes.reset.statuses.enabledStatus.disabled
        OnMouseClick: execute { ref.processes.reset.do_request := TRUE; }
    Frame (30,325 205x20)
        shows VISU_StatusWidget(widget := widget.processes_resetStatus)
        p4168582468: ref.processes.reset.actualStatus
    Frame (30,235 205x20)
        shows VISU_StatusWidget(widget := widget.processes_doHomingStatus)
        p4168582468: ref.processes.doHoming.actualStatus
    Button (30,445 205x60), "QuickStop axes", input disabled if: ref.processes.quickStop.statuses.enabledStatus.disabled
        OnMouseClick: execute { ref.processes.quickStop.do_request := TRUE; }
    Frame (30,420 205x20)
        shows VISU_StatusWidget(widget := widget.processes_quickStopStatus)
        p4168582468: ref.processes.quickStop.actualStatus
    Label (305,235 40x20), "AZI"
    Rectangle (345,235 95x20), "%.1f Nm", text variable: ref.parts.azi.actTorqueAzi.newtonmeter.value
    Label (305,255 40x20), "ABL"
    Rectangle (345,255 95x20), "%.1f Nm", text variable: ref.parts.azi.actTorqueAbl.newtonmeter.value
    Label (305,275 40x20), "ELE"
    Rectangle (345,275 95x20), "%.1f Nm", text variable: ref.parts.ele.actTorque.newtonmeter.value
    Label (305,295 40x20), "ROC"
    Rectangle (345,295 95x20), "%.1f Nm", text variable: ref.parts.roc.actTorque.newtonmeter.value
    Label (305,315 40x20), "RON"
    Rectangle (345,315 95x20), "%.1f Nm", text variable: ref.parts.ron.actTorque.newtonmeter.value
    Polyline (390,215) (470,215) (470,345) (285,345) (285,215) (310,215)
    Label (315,205 60x20), "Torque"
END_VISUALIZATION

// ---- MTCS/Axes/Visu/VISU_AxesPointingModelConfig_part1.TcVIS
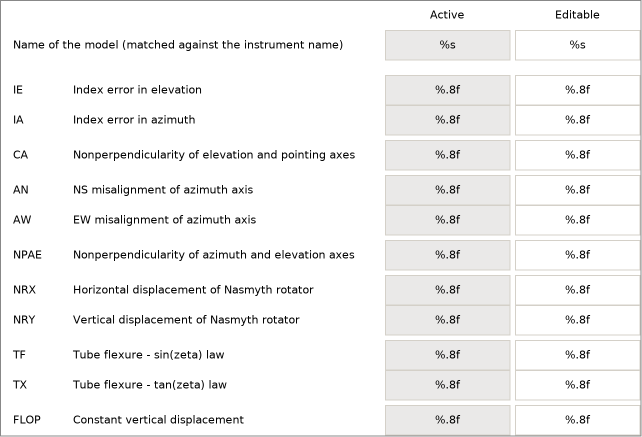
VISUALIZATION VISU_AxesPointingModelConfig_part1  // 642x437
VAR_IN_OUT
    active : AxesPointingModelConfig;
    editable : AxesPointingModelConfig;
END_VAR
    Label (385,5 125x20), "Active"
    Label (515,5 125x20), "Editable"
    Label (10,75 30x30), "IE"
    Frame (385,75 255x30)
        shows VISU_ConfigLREAL8Entry(active := active.IE, editable := editable.IE)
    Label (70,75 315x30), "Index error in elevation"
    Label (10,105 30x30), "IA"
    Frame (385,105 255x30)
        shows VISU_ConfigLREAL8Entry(active := active.IA, editable := editable.IA)
    Label (70,105 315x30), "Index error in azimuth"
    Label (10,140 30x30), "CA"
    Frame (385,140 255x30)
        shows VISU_ConfigLREAL8Entry(active := active.CA, editable := editable.CA)
    Label (70,140 315x30), "Nonperpendicularity of elevation and pointing axes"
    Label (10,175 30x30), "AN"
    Frame (385,175 255x30)
        shows VISU_ConfigLREAL8Entry(active := active.AN, editable := editable.AN)
    Label (70,175 315x30), "NS misalignment of azimuth axis"
    Frame (385,205 255x30)
        shows VISU_ConfigLREAL8Entry(active := active.AW, editable := editable.AW)
    Label (10,205 60x30), "AW"
    Label (70,205 315x30), "EW misalignment of azimuth axis"
    Frame (385,240 255x30)
        shows VISU_ConfigLREAL8Entry(active := active.NPAE, editable := editable.NPAE)
    Label (10,240 60x30), "NPAE"
    Label (70,240 315x30), "Nonperpendicularity of azimuth and elevation axes"
    Frame (385,275 255x30)
        shows VISU_ConfigLREAL8Entry(active := active.NRX, editable := editable.NRX)
    Label (10,275 60x30), "NRX"
    Label (70,275 315x30), "Horizontal displacement of Nasmyth rotator"
    Frame (385,305 255x30)
        shows VISU_ConfigLREAL8Entry(active := active.NRY, editable := editable.NRY)
    Label (10,305 60x30), "NRY"
    Label (70,305 315x30), "Vertical displacement of Nasmyth rotator"
    Frame (385,340 255x30)
        shows VISU_ConfigLREAL8Entry(active := active.TF, editable := editable.TF)
    Label (10,340 60x30), "TF"
    Label (70,340 315x30), "Tube flexure - sin(zeta) law"
    Frame (385,370 255x30)
        shows VISU_ConfigLREAL8Entry(active := active.TX, editable := editable.TX)
    Label (10,370 60x30), "TX"
    Label (70,370 315x30), "Tube flexure - tan(zeta) law"
    Frame (385,30 255x30)
        shows VISU_ConfigStringEntry(active := active.name, editable := editable.name)
    Label (10,30 370x30), "Name of the model (matched against the instrument name)"
    Frame (385,405 255x30)
        shows VISU_ConfigLREAL8Entry(active := active.FLOP, editable := editable.FLOP)
    Label (10,405 60x30), "FLOP"
    Label (70,405 315x30), "Constant vertical displacement"
END_VISUALIZATION

// ---- MTCS/Axes/Visu/VISU_AxesPointingModelConfig_part2.TcVIS
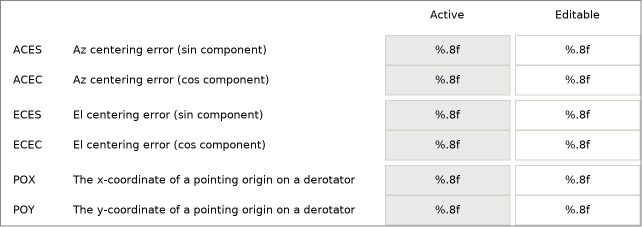
VISUALIZATION VISU_AxesPointingModelConfig_part2  // 642x227
VAR_IN_OUT
    active : AxesPointingModelConfig;
    editable : AxesPointingModelConfig;
END_VAR
    Label (385,5 125x20), "Active"
    Label (515,5 125x20), "Editable"
    Label (10,35 50x30), "ACES"
    Frame (385,35 255x30)
        shows VISU_ConfigLREAL8Entry(active := active.ACES, editable := editable.ACES)
    Label (70,35 315x30), "Az centering error (sin component)"
    Label (10,65 50x30), "ACEC"
    Frame (385,65 255x30)
        shows VISU_ConfigLREAL8Entry(active := active.ACEC, editable := editable.ACEC)
    Label (70,65 315x30), "Az centering error (cos component)"
    Label (10,100 50x30), "ECES"
    Frame (385,100 255x30)
        shows VISU_ConfigLREAL8Entry(active := active.ECES, editable := editable.ECES)
    Label (70,100 315x30), "El centering error (sin component)"
    Label (10,130 50x30), "ECEC"
    Frame (385,130 255x30)
        shows VISU_ConfigLREAL8Entry(active := active.ECEC, editable := editable.ECEC)
    Label (70,130 315x30), "El centering error (cos component)"
    Label (10,165 50x30), "POX"
    Frame (385,165 255x30)
        shows VISU_ConfigLREAL8Entry(active := active.POX, editable := editable.POX)
    Label (70,165 315x30), "The x-coordinate of a pointing origin on a derotator"
    Label (10,195 50x30), "POY"
    Frame (385,195 255x30)
        shows VISU_ConfigLREAL8Entry(active := active.POY, editable := editable.POY)
    Label (70,195 315x30), "The y-coordinate of a pointing origin on a derotator"
END_VISUALIZATION

// ---- MTCS/Axes/Visu/VISU_AxesPointingModelSetup.TcVIS
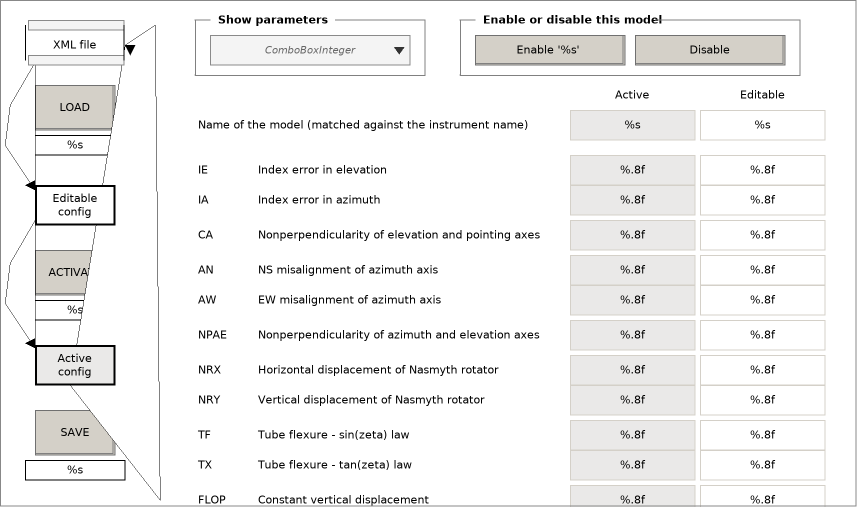
VISUALIZATION VISU_AxesPointingModelSetup  // 857x507
VAR_IN_OUT
    ref : AxesPointingModelSetup;
    widget : AxesPointingModelSetupWidget;
END_VAR
    Polyline (210,20) (195,20) (195,75) (425,75) (425,20) (335,20)
    Frame (10,10 180x495)
        shows VISU_ConfigManager(mgr := ref.parts.configManager, widget := widget.configManager)
    Frame (185,80 670x420), frame switch variable: widget.part
        shows VISU_AxesPointingModelConfig_part1(active := ref.config, editable := ref.editableConfig)
        shows VISU_AxesPointingModelConfig_part2(active := ref.config, editable := ref.editableConfig)
        shows VISU_MeasurementConfig(active := active.temperatures.m2Electronics, editable := editable.temperatures.m2Electronics)
        shows VISU_MeasurementConfig(active := active.temperatures.topTube, editable := editable.temperatures.topTube)
        shows VISU_MeasurementConfig(active := active.temperatures.centreTube, editable := editable.temperatures.centreTube)
        shows VISU_MeasurementConfig(active := active.temperatures.fork, editable := editable.temperatures.fork)
        shows VISU_MeasurementConfig(active := active.temperatures.nasmythAir, editable := editable.temperatures.nasmythAir)
        shows VISU_MeasurementConfig(active := active.temperatures.rem, editable := editable.temperatures.rem)
        shows VISU_MeasurementConfig(active := active.temperatures.rpm, editable := editable.temperatures.rpm)
        shows VISU_MeasurementConfig(active := active.temperatures.hermesTelescopeAdapter, editable := editable.temperatures.hermesTelescopeAdapter)
        shows VISU_MeasurementConfig(active := active.temperatures.topAir, editable := editable.temperatures.topAir)
        shows VISU_MeasurementConfig(active := active.temperatures.insideTube, editable := editable.temperatures.insideTube)
        shows VISU_MeasurementConfig(active := active.relativeHumidities.topAir, editable := editable.relativeHumidities.topAir)
        shows VISU_MeasurementConfig(active := active.relativeHumidities.insideTube, editable := editable.relativeHumidities.insideTube)
        shows VISU_MeasurementConfig(active := active.dewpoints.topAir, editable := editable.dewpoints.topAir)
        shows VISU_MeasurementConfig(active := active.dewpoints.insideTube, editable := editable.dewpoints.insideTube)
        shows VISU_MeasurementConfig(active := active.accelerometers.tube.x, editable := editable.accelerometers.tube.x)
        shows VISU_MeasurementConfig(active := active.accelerometers.tube.y, editable := editable.accelerometers.tube.y)
        shows VISU_AxesConfig_LocalConditions(active := active.localConditions, editable := editable.localConditions)
    ComboBoxInteger (210,35 200x30), variable: widget.part, text list: 'AxesPointingModelSetupPartsTextList'
    Label (480,10 180x20), "Enable or disable this model"
    Polyline (475,20) (460,20) (460,75) (800,75) (800,20) (655,20)
    Button (475,35 150x30), "Enable '%s'", text variable: ref.config.name, input disabled if: widget.enableButtonDisabled
        OnMouseClick: execute { widget.enableButtonPressed := TRUE; }
    Button (635,35 150x30), "Disable", input disabled if: widget.disableButtonDisabled
        OnMouseClick: execute { widget.disableButtonPressed := TRUE; }
    Label (215,10 125x20), "Show parameters"
END_VISUALIZATION

// ---- MTCS/Axes/Visu/VISU_AxesConfig_General.TcVIS
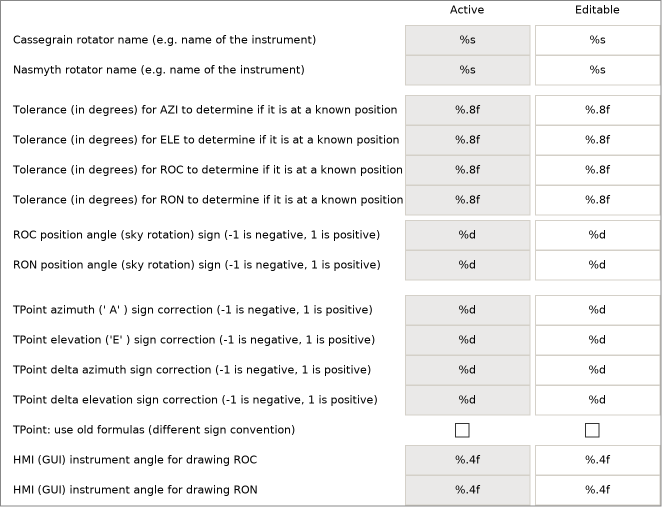
VISUALIZATION VISU_AxesConfig_General  // 662x507
VAR_IN_OUT
    editable : AxesConfig;
	active : AxesConfig;
END_VAR
    Frame (405,25 255x30)
        shows VISU_ConfigStringEntry(active := active.cassegrainRotatorName, editable := editable.cassegrainRotatorName)
    Label (405,0 125x20), "Active"
    Label (535,0 125x20), "Editable"
    Label (10,25 370x30), "Cassegrain rotator name (e.g. name of the instrument)"
    Frame (405,55 255x30)
        shows VISU_ConfigStringEntry(active := active.nasmythRotatorName, editable := editable.nasmythRotatorName)
    Label (10,55 370x30), "Nasmyth rotator name (e.g. name of the instrument)"
    Frame (405,95 255x30)
        shows VISU_ConfigLREAL8Entry(active := active.knownPositionToleranceAzi, editable := editable.knownPositionToleranceAzi)
    Label (10,95 395x30), "Tolerance (in degrees) for AZI to determine if it is at a known position"
    Label (10,125 395x30), "Tolerance (in degrees) for ELE to determine if it is at a known position"
    Frame (405,125 255x30)
        shows VISU_ConfigLREAL8Entry(active := active.knownPositionToleranceEle, editable := editable.knownPositionToleranceEle)
    Label (10,155 395x30), "Tolerance (in degrees) for ROC to determine if it is at a known position"
    Frame (405,155 255x30)
        shows VISU_ConfigLREAL8Entry(active := active.knownPositionToleranceRoc, editable := editable.knownPositionToleranceRoc)
    Label (10,185 395x30), "Tolerance (in degrees) for RON to determine if it is at a known position"
    Frame (405,185 255x30)
        shows VISU_ConfigLREAL8Entry(active := active.knownPositionToleranceRon, editable := editable.knownPositionToleranceRon)
    Frame (405,295 255x30)
        shows VISU_ConfigINTEntry(active := active.tpointAziSign, editable := editable.tpointAziSign)
    Label (10,295 395x30), "TPoint azimuth (' A' ) sign correction (-1 is negative, 1 is positive)"
    Frame (405,325 255x30)
        shows VISU_ConfigINTEntry(active := active.tpointEleSign, editable := editable.tpointEleSign)
    Label (10,325 395x30), "TPoint elevation ('E' ) sign correction (-1 is negative, 1 is positive)"
    Frame (405,355 255x30)
        shows VISU_ConfigINTEntry(active := active.tpointDeltaAziSign, editable := editable.tpointDeltaAziSign)
    Label (10,355 395x30), "TPoint delta azimuth sign correction (-1 is negative, 1 is positive)"
    Frame (405,385 255x30)
        shows VISU_ConfigINTEntry(active := active.tpointDeltaEleSign, editable := editable.tpointDeltaEleSign)
    Label (10,385 395x30), "TPoint delta elevation sign correction (-1 is negative, 1 is positive)"
    Label (10,415 395x30), "TPoint: use old formulas (different sign convention)"
    Frame (405,415 255x30)
        shows VISU_ConfigBOOLEntry(active := active.tpointOldFormulas, editable := editable.tpointOldFormulas)
    Frame (405,220 255x30)
        shows VISU_ConfigINTEntry(active := active.rocPositionAngleSign, editable := editable.rocPositionAngleSign)
    Label (10,220 395x30), "ROC position angle (sky rotation) sign (-1 is negative, 1 is positive)"
    Frame (405,250 255x30)
        shows VISU_ConfigINTEntry(active := active.ronPositionAngleSign, editable := editable.ronPositionAngleSign)
    Label (10,250 395x30), "RON position angle (sky rotation) sign (-1 is negative, 1 is positive)"
    Frame (405,445 255x30)
        shows VISU_ConfigLREAL4Entry(active := active.rocGuiAngle, editable := editable.rocGuiAngle)
    Label (10,445 395x30), "HMI (GUI) instrument angle for drawing ROC"
    Frame (405,475 255x30)
        shows VISU_ConfigLREAL4Entry(active := active.ronGuiAngle, editable := editable.ronGuiAngle)
    Label (10,475 395x30), "HMI (GUI) instrument angle for drawing RON"
END_VISUALIZATION

// ---- MTCS/Axes/Visu/VISU_AxesConfig_Location.TcVIS
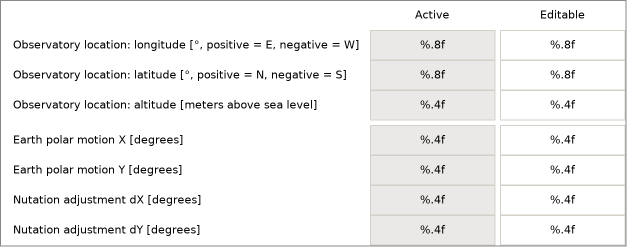
VISUALIZATION VISU_AxesConfig_Location  // 627x247
VAR_IN_OUT
    active : AxesLocationConfig;
    editable : AxesLocationConfig;
END_VAR
    Label (370,5 125x20), "Active"
    Label (500,5 125x20), "Editable"
    Label (10,30 360x30), "Observatory location: longitude [°, positive = E, negative = W]"
    Frame (370,30 255x30)
        shows VISU_ConfigLREAL8Entry(active := active.longitude, editable := editable.longitude)
    Frame (370,60 255x30)
        shows VISU_ConfigLREAL8Entry(active := active.latitude, editable := editable.latitude)
    Label (10,60 360x30), "Observatory location: latitude [°, positive = N, negative = S]"
    Label (10,90 360x30), "Observatory location: altitude [meters above sea level]"
    Frame (370,90 255x30)
        shows VISU_ConfigREAL4Entry(active := active.height, editable := editable.height)
    Label (10,125 360x30), "Earth polar motion X [degrees]"
    Frame (370,125 255x30)
        shows VISU_ConfigREAL4Entry(active := active.polarMotionX, editable := editable.polarMotionX)
    Label (10,155 360x30), "Earth polar motion Y [degrees]"
    Frame (370,155 255x30)
        shows VISU_ConfigREAL4Entry(active := active.polarMotionY, editable := editable.polarMotionY)
    Frame (370,185 255x30)
        shows VISU_ConfigREAL4Entry(active := active.nutationDx, editable := editable.nutationDx)
    Label (10,185 360x30), "Nutation adjustment dX [degrees]"
    Label (10,215 360x30), "Nutation adjustment dY [degrees]"
    Frame (370,215 255x30)
        shows VISU_ConfigREAL4Entry(active := active.nutationDy, editable := editable.nutationDy)
END_VISUALIZATION

// ---- MTCS/Axes/Visu/VISU_AxesConfig_LocalConditions.TcVIS
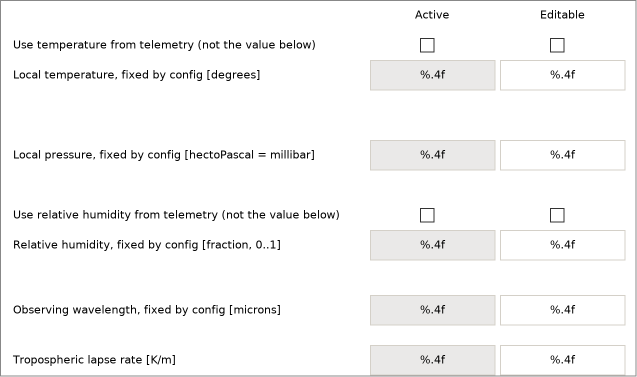
VISUALIZATION VISU_AxesConfig_LocalConditions  // 637x377
VAR_IN_OUT
    active : AxesLocalConditionsConfig;
    editable : AxesLocalConditionsConfig;
END_VAR
    Label (370,5 125x20), "Active"
    Label (500,5 125x20), "Editable"
    Label (10,30 360x30), "Use temperature from telemetry (not the value below)"
    Frame (370,30 265x30)
        shows VISU_ConfigBOOLEntry(active := active.useTemperatureFromSensors, editable := editable.useTemperatureFromSensors)
    Label (10,60 360x30), "Local temperature, fixed by config [degrees]"
    Frame (370,60 255x30)
        shows VISU_ConfigREAL4Entry(active := active.configuredTemperature, editable := editable.configuredTemperature)
    Label (10,140 360x30), "Local pressure, fixed by config [hectoPascal = millibar]"
    Frame (370,140 255x30)
        shows VISU_ConfigREAL4Entry(active := active.configuredPressure, editable := editable.configuredPressure)
    Label (10,230 360x30), "Relative humidity, fixed by config [fraction, 0..1]"
    Label (10,200 360x30), "Use relative humidity from telemetry (not the value below)"
    Frame (370,200 265x30)
        shows VISU_ConfigBOOLEntry(active := active.useRelativeHumidityFromSensors, editable := editable.useRelativeHumidityFromSensors)
    Frame (370,230 255x30)
        shows VISU_ConfigREAL4Entry(active := active.configuredRelativeHumidity, editable := editable.configuredRelativeHumidity)
    Label (10,295 360x30), "Observing wavelength, fixed by config [microns]"
    Frame (370,295 255x30)
        shows VISU_ConfigREAL4Entry(active := active.configuredObservingWavelength, editable := editable.configuredObservingWavelength)
    Label (10,345 360x30), "Tropospheric lapse rate [K/m]"
    Frame (370,345 255x30)
        shows VISU_ConfigREAL4Entry(active := active.troposphericLapseRate, editable := editable.troposphericLapseRate)
END_VISUALIZATION

// ---- MTCS/Axes/Visu/VISU_AxesFromCpp_Target.TcVIS
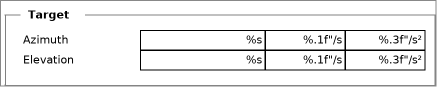
VISUALIZATION VISU_AxesFromCpp_Target  // 437x87
VAR_IN_OUT
	ref : Axes;
    widget : AxesWidget;
END_VAR
    Polyline (20,15) (5,15) (5,85) (435,85) (435,15) (85,15)
    Label (25,5 60x20), "Target"
    Label (20,30 80x20), "Azimuth"
    Label (20,50 80x20), "Elevation"
    Rectangle (140,30 125x20), "%s", text variable: widget.axes.azi.targetPos.dmsString
    Rectangle (140,50 125x20), "%s", text variable: widget.axes.ele.targetPos.dmsString
    Rectangle (265,30 80x20), "%.1f"/s", text variable: ref.target.aziVelo.arcsecondsPerSecond.value
    Rectangle (345,30 80x20), "%.3f"/s²", text variable: ref.target.aziAcc.arcsecondsPerSquareSecond.value
    Rectangle (345,50 80x20), "%.3f"/s²", text variable: ref.target.eleAcc.arcsecondsPerSquareSecond.value
    Rectangle (265,50 80x20), "%.1f"/s", text variable: ref.target.eleVelo.arcsecondsPerSecond.value
END_VISUALIZATION

// ---- MTCS/Axes/Visu/VISU_AxesIO.TcVIS
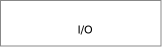
VISUALIZATION VISU_AxesIO  // 162x47
VAR_IN_OUT
	ref : AxesIO;
    widget : AxesIOWidget;
END_VAR
    Label (10,15 150x30), "I/O"
END_VISUALIZATION

// ---- MTCS/Axes/Visu/VISU_Axes.TcVIS
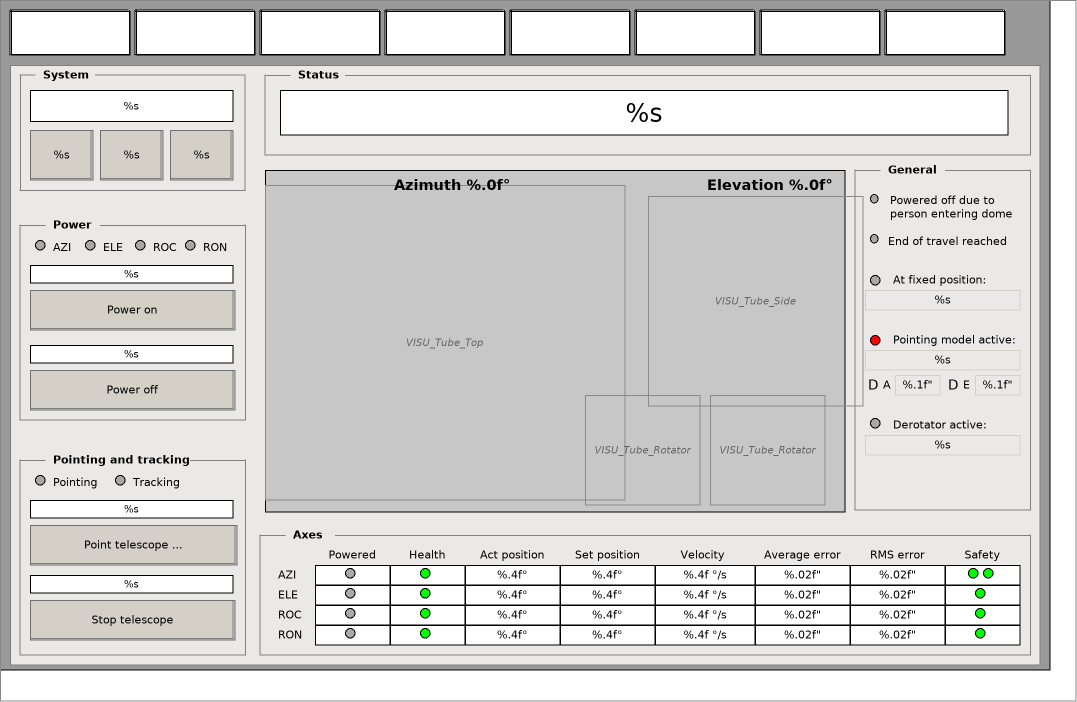
VISUALIZATION VISU_Axes  // 1077x702
VAR_IN_OUT
	ref : Axes;
    widget : AxesWidget;
END_VAR
    Frame (0,0 1075x700)
        shows VISU_SystemBackground(color := widget.actualStatus.color)
    Frame (10,60 1035x605)
        shows VISU_AxesOverview(ref := ref, widget := widget)
        shows VISU_AxesManual(ref := ref, widget := widget.manual)
        shows VISU_AxesAxes(ref := ref, widget := widget.axes)
        shows VISU_AxesTarget(ref := ref, widget := widget)
        shows VISU_AxesPointingModelsSetup(ref := ref.parts.tpoint, widget := widget.tpoint)
        shows VISU_AxesAdvanced(ref := ref, widget := widget)
        shows VISU_AxesIO(ref := ref.parts.io, widget := widget.io)
        shows VISU_AxesConfig(editable := ref.editableConfig, active := ref.config, mgr := ref.parts.configManager, mgrWidget := widget.configManager, axesWidget := widget)
        p701045219: ref.editableConfig
        p2690442461: ref.config
        p942769723: ref.parts.configManager
        p2963374678: widget.configManager
        p459268616: widget
        p4094514409: widget
        p1371549466: ref.editableConfig
        p1340763843: ref.config
        p2803088772: widget
        p2427492753: ref.parts.aziDrive
        p1656878407: ref.parts.ablDrive
        p2190985393: ref.parts.eleDrive
    Frame (10,10 120x50)
        shows VISU_SubSystemButton(widget := widget.button_overview)
        OnMouseClick: FrameSelectionChange Selection=SelectedFrame=b1e9e4b0-bf3d-440f-90c5-cb513105ccf1, GlobSel=AssignType=Directly, SelType=Locally
        OnMouseClick: execute { widget.activeTab := AxesTabs.OVERVIEW; }
    Frame (635,10 120x50)
        shows VISU_SubSystemButton(widget := widget.button_advanced)
        OnMouseClick: FrameSelectionChange Selection=SelectedFrame=b1e9e4b0-bf3d-440f-90c5-cb513105ccf1, Selection=5, GlobSel=AssignType=Directly, SelType=Locally
        OnMouseClick: execute { widget.activeTab := AxesTabs.ADVANCED; }
    Frame (760,10 120x50)
        shows VISU_SubSystemButton(widget := widget.button_io)
        OnMouseClick: FrameSelectionChange Selection=SelectedFrame=b1e9e4b0-bf3d-440f-90c5-cb513105ccf1, Selection=6, GlobSel=AssignType=Directly, SelType=Locally
        OnMouseClick: execute { widget.activeTab := AxesTabs.IO; }
    Frame (135,10 120x50)
        shows VISU_SubSystemButton(widget := widget.button_manual)
        OnMouseClick: FrameSelectionChange Selection=SelectedFrame=b1e9e4b0-bf3d-440f-90c5-cb513105ccf1, Selection=1, GlobSel=AssignType=Directly, SelType=Locally
        OnMouseClick: execute { widget.activeTab := AxesTabs.MANUAL; }
    Frame (260,10 120x50)
        shows VISU_SubSystemButton(widget := widget.button_axes)
        OnMouseClick: FrameSelectionChange Selection=SelectedFrame=b1e9e4b0-bf3d-440f-90c5-cb513105ccf1, Selection=2, GlobSel=AssignType=Directly, SelType=Locally
        OnMouseClick: execute { widget.activeTab := AxesTabs.AXES; }
    Frame (385,10 120x50)
        shows VISU_SubSystemButton(widget := widget.button_target)
        OnMouseClick: FrameSelectionChange Selection=SelectedFrame=b1e9e4b0-bf3d-440f-90c5-cb513105ccf1, Selection=3, GlobSel=AssignType=Directly, SelType=Locally
        OnMouseClick: execute { widget.activeTab := AxesTabs.TARGET; }
    Frame (510,10 120x50)
        shows VISU_SubSystemButton(widget := widget.button_tpoint)
        OnMouseClick: FrameSelectionChange Selection=SelectedFrame=b1e9e4b0-bf3d-440f-90c5-cb513105ccf1, Selection=4, GlobSel=AssignType=Directly, SelType=Locally
        OnMouseClick: execute { widget.activeTab := AxesTabs.TPOINT; }
    Frame (885,10 120x50)
        shows VISU_SubSystemButton(widget := widget.button_config)
        OnMouseClick: FrameSelectionChange Selection=SelectedFrame=b1e9e4b0-bf3d-440f-90c5-cb513105ccf1, Selection=7, GlobSel=AssignType=Directly, SelType=Locally
        OnMouseClick: execute { widget.activeTab := AxesTabs.CONFIG; }
END_VISUALIZATION

// ---- MTCS/Axes/Visu/VISU_AxesOverview.TcVIS
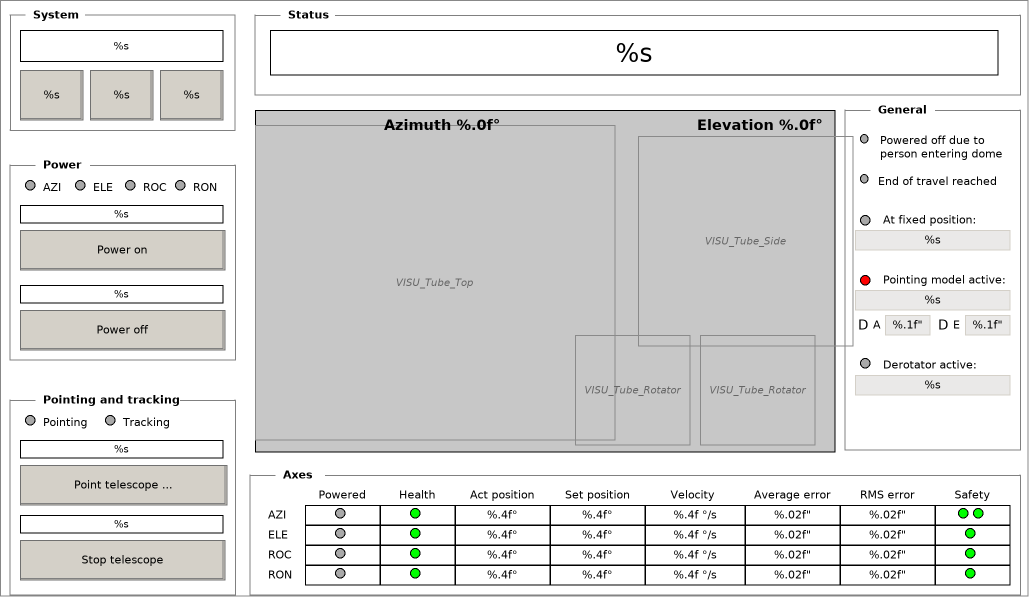
VISUALIZATION VISU_AxesOverview  // 1029x597
VAR_IN_OUT
	ref : Axes;
    widget : AxesWidget;
END_VAR
    Polyline (935,110) (1020,110) (1020,450) (845,450) (845,110) (870,110)
    Frame (255,110 598x342)
        shows VISU_AxesImage(ref := ref, widget := widget)
    Polyline (180,400) (235,400) (235,595) (10,595) (10,400) (35,400)
    Polyline (90,165) (235,165) (235,360) (10,360) (10,165) (35,165)
    Frame (10,5 226x126)
        shows VISU_SystemControl(status := widget.actualStatus, button_initialize := widget.button_initialize, button_operating := widget.button_operating, button_locking := widget.button_locking)
    Button (20,230 205x40), "Power on", input disabled if: ref.processes.powerOn.statuses.enabledStatus.disabled
        OnMouseClick: execute {
            ref.processes.powerOn.request(
                azi := TRUE,
                ele := TRUE,
                roc := FALSE,
                ron := FALSE,
                fw := FALSE);
        }
    Button (20,540 205x40), "Stop telescope", input disabled if: ref.processes.stop.statuses.enabledStatus.disabled
        OnMouseClick: execute { ref.processes.stop.do_request := TRUE; }
    Button (20,310 205x40), "Power off", input disabled if: ref.processes.powerOff.statuses.enabledStatus.disabled
        OnMouseClick: execute { ref.processes.powerOff.do_request := TRUE; }
    Frame (25,175 10x15)
        shows VISU_State_gray_green(state := ref.parts.azi.statuses.poweredStatus.enabled)
    Label (40,175 30x25), "AZI"
    Button (20,465 207x40), "Point telescope ..."
        OnMouseClick: OpenDialog Dialog=VISU_AxesPointDialog, OpenModal=True, OpenCentered=True
    Frame (860,130 10x15)
        shows VISU_State_gray_orange(state := ref.isPoweredOffByPersonInDome)
    Label (877,132 150x30), "Powered off due to person entering dome"
    Rectangle (855,230 155x20), "%s", text variable: ref.actualKnownPositionName, colour toggle: ref.isAtKnownPosition
    Label (880,205 125x30), "At fixed position:"
    Rectangle (855,290 155x20), "%s", text variable: widget.activePointingModelString
    Label (880,265 140x30), "Pointing model active:"
    Rectangle (855,375 155x20), "%s", text variable: widget.activeRotatorString
    Label (880,355 125x20), "Derotator active:"
    Label (40,155 50x20), "Power"
    Frame (20,515 205x20)
        shows VISU_StatusWidget(widget := widget.processes_stopStatus)
        p4168582468: ref.processes.stop.actualStatus
    Frame (20,440 205x20)
        shows VISU_StatusWidget(widget := widget.processes_pointStatus)
        p4168582468: ref.processes.point.actualStatus
    Frame (20,285 205x20)
        shows VISU_StatusWidget(widget := widget.processes_powerOffStatus)
        p4168582468: ref.processes.reset.actualStatus
    Frame (20,205 205x20)
        shows VISU_StatusWidget(widget := widget.processes_powerOnStatus)
        p4168582468: ref.processes.reset.actualStatus
    Label (40,390 135x20), "Pointing and tracking"
    Frame (75,175 10x15)
        shows VISU_State_gray_green(state := ref.parts.ele.statuses.poweredStatus.enabled)
    Label (90,175 30x25), "ELE"
    Frame (125,175 10x15)
        shows VISU_State_gray_green(state := ref.parts.roc.statuses.poweredStatus.enabled)
    Label (140,175 30x25), "ROC"
    Frame (175,175 10x15)
        shows VISU_State_gray_green(state := ref.parts.ron.statuses.poweredStatus.enabled)
    Label (190,175 30x25), "RON"
    Frame (25,410 10x15)
        shows VISU_State_gray_green(state := ref.isPointing)
    Label (40,410 60x25), "Pointing"
    Label (120,410 60x25), "Tracking"
    Frame (105,410 10x15)
        shows VISU_State_gray_green(state := ref.isTracking)
    Frame (860,270 5x12)
        shows VISU_State_red_green(state := ref.isPointingModelActive)
    Frame (860,210 15x15)
        shows VISU_State_gray_green(state := ref.isAtKnownPosition)
    Frame (860,353 15x15)
        shows VISU_State_gray_green(state := widget.isDerotatorActive)
    Label (870,315 15x20), "A"
    Label (855,315 20x20), "D"
    Rectangle (885,315 45x20), "%.1f"", text variable: ref.target.aziPointingModelOffset.arcseconds.value
    Label (950,315 15x20), "E"
    Label (935,315 20x20), "D"
    Rectangle (965,315 45x20), "%.1f"", text variable: ref.target.elePointingModelOffset.arcseconds.value
    Frame (860,170 10x15)
        shows VISU_State_gray_red(state := ref.isLimitsReached)
    Label (875,170 150x23), "End of travel reached"
    Polyline (335,15) (1020,15) (1020,95) (255,95) (255,15) (280,15)
    Label (285,5 50x20), "Status"
    Frame (270,30 735x50)
        shows VISU_StatusWidget(widget := widget.actualStatus)
        p4168582468: ref.processes.reset.actualStatus
    Polyline (325,475) (1020,475) (1020,595) (250,595) (250,475) (275,475)
    Label (280,465 70x20), "Axes"
    Frame (260,480 515x105)
        shows VISU_Axes_stats(ref := ref, widget := widget)
    Label (875,100 70x20), "General"
END_VISUALIZATION

// ---- MTCS/Axes/Visu/VISU_AxesMultiMoveProcess.TcVIS
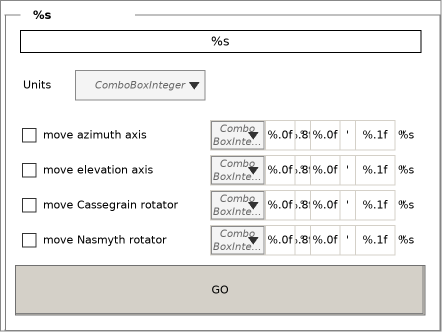
VISUALIZATION VISU_AxesMultiMoveProcess  // 442x332
VAR_IN_OUT
	ref : AxesMultiMoveProcess;
    widget : AxesMultiMoveProcessWidget;
END_VAR
    Polyline (20,15) (5,15) (5,330) (440,330) (440,15) (135,15)
    Label (20,70 80x30), "Units"
    ComboBoxInteger (75,70 130x30), variable: widget.units, text list: 'AxesMoveProcessUnitsTextList'
    Rectangle (395,120 35x30), "%s", text variable: widget.unitsText, invisible if: widget.units = AxesMoveProcessWidgetUnits.DEGMINSEC
    Checkbox (20,120 180x30), "move azimuth axis", variable: widget.selected_azi
    Textfield (210,120 180x30), "%.8f", text variable: widget.field_azi_decimal, invisible if: widget.units = AxesMoveProcessWidgetUnits.DEGMINSEC
        OnMouseClick: write the text variable via VisuDialogs.Numpad
    Textfield (265,120 30x30), "%.0f", text variable: widget.field_azi_d, invisible if: widget.units <> AxesMoveProcessWidgetUnits.DEGMINSEC
        OnMouseClick: write the text variable via VisuDialogs.Numpad
    ComboBoxInteger (211,121 53x28), variable: widget.field_azi_sign, invisible if: widget.units <> AxesMoveProcessWidgetUnits.DEGMINSEC, text list: 'AxesDialogSignTextList'
    Textfield (310,120 30x30), "%.0f", text variable: widget.field_azi_m, invisible if: widget.units <> AxesMoveProcessWidgetUnits.DEGMINSEC
        OnMouseClick: write the text variable via VisuDialogs.Numpad
    Textfield (355,120 40x30), "%.1f", text variable: widget.field_azi_s, invisible if: widget.units <> AxesMoveProcessWidgetUnits.DEGMINSEC
        OnMouseClick: write the text variable via VisuDialogs.Numpad
    Label (295,120 15x30), "°", invisible if: widget.units <> AxesMoveProcessWidgetUnits.DEGMINSEC
    Label (340,120 15x30), "'", invisible if: widget.units <> AxesMoveProcessWidgetUnits.DEGMINSEC
    Label (395,120 15x30), """, invisible if: widget.units <> AxesMoveProcessWidgetUnits.DEGMINSEC
    Button (15,265 410x50), "GO", input disabled if: ref.statuses.enabledStatus.disabled
        OnMouseClick: execute {
            ref.request(
                units := AxesMoveUnits.DEGREES,
                azi := widget.aziDeg,
                ele := widget.eleDeg,
                rot := 0.0,
                roc := widget.rocDeg,
                ron := widget.ronDeg,
                doAzi := widget.selected_azi,
                doEle := widget.selected_ele,
                doRot := FALSE,
                doRoc := widget.selected_roc,
                doRon := widget.selected_ron,
                preferMostTravel := FALSE);
        }
    Checkbox (20,190 185x30), "move Cassegrain rotator", variable: widget.selected_roc
    Checkbox (20,225 175x30), "move Nasmyth rotator", variable: widget.selected_ron
    Checkbox (20,155 180x30), "move elevation axis", variable: widget.selected_ele
    Rectangle (395,155 35x30), "%s", text variable: widget.unitsText, invisible if: widget.units = AxesMoveProcessWidgetUnits.DEGMINSEC
    Textfield (210,155 180x30), "%.8f", text variable: widget.field_ele_decimal, invisible if: widget.units = AxesMoveProcessWidgetUnits.DEGMINSEC
        OnMouseClick: write the text variable via VisuDialogs.Numpad
    Textfield (265,155 30x30), "%.0f", text variable: widget.field_ele_d, invisible if: widget.units <> AxesMoveProcessWidgetUnits.DEGMINSEC
        OnMouseClick: write the text variable via VisuDialogs.Numpad
    ComboBoxInteger (211,156 53x28), variable: widget.field_ele_sign, invisible if: widget.units <> AxesMoveProcessWidgetUnits.DEGMINSEC, text list: 'AxesDialogSignTextList'
    Textfield (310,155 30x30), "%.0f", text variable: widget.field_ele_m, invisible if: widget.units <> AxesMoveProcessWidgetUnits.DEGMINSEC
        OnMouseClick: write the text variable via VisuDialogs.Numpad
    Textfield (355,155 40x30), "%.1f", text variable: widget.field_ele_s, invisible if: widget.units <> AxesMoveProcessWidgetUnits.DEGMINSEC
        OnMouseClick: write the text variable via VisuDialogs.Numpad
    Label (295,155 15x30), "°", invisible if: widget.units <> AxesMoveProcessWidgetUnits.DEGMINSEC
    Label (340,155 15x30), "'", invisible if: widget.units <> AxesMoveProcessWidgetUnits.DEGMINSEC
    Label (395,155 15x30), """, invisible if: widget.units <> AxesMoveProcessWidgetUnits.DEGMINSEC
    Rectangle (395,190 35x30), "%s", text variable: widget.unitsText, invisible if: widget.units = AxesMoveProcessWidgetUnits.DEGMINSEC
    Textfield (210,190 180x30), "%.8f", text variable: widget.field_roc_decimal, invisible if: widget.units = AxesMoveProcessWidgetUnits.DEGMINSEC
        OnMouseClick: write the text variable via VisuDialogs.Numpad
    Textfield (265,190 30x30), "%.0f", text variable: widget.field_roc_d, invisible if: widget.units <> AxesMoveProcessWidgetUnits.DEGMINSEC
        OnMouseClick: write the text variable via VisuDialogs.Numpad
    ComboBoxInteger (211,191 53x28), variable: widget.field_roc_sign, invisible if: widget.units <> AxesMoveProcessWidgetUnits.DEGMINSEC, text list: 'AxesDialogSignTextList'
    Textfield (310,190 30x30), "%.0f", text variable: widget.field_roc_m, invisible if: widget.units <> AxesMoveProcessWidgetUnits.DEGMINSEC
        OnMouseClick: write the text variable via VisuDialogs.Numpad
    Textfield (355,190 40x30), "%.1f", text variable: widget.field_roc_s, invisible if: widget.units <> AxesMoveProcessWidgetUnits.DEGMINSEC
        OnMouseClick: write the text variable via VisuDialogs.Numpad
    Label (295,190 15x30), "°", invisible if: widget.units <> AxesMoveProcessWidgetUnits.DEGMINSEC
    Label (340,190 15x30), "'", invisible if: widget.units <> AxesMoveProcessWidgetUnits.DEGMINSEC
    Label (395,190 15x30), """, invisible if: widget.units <> AxesMoveProcessWidgetUnits.DEGMINSEC
    Rectangle (395,225 35x30), "%s", text variable: widget.unitsText, invisible if: widget.units = AxesMoveProcessWidgetUnits.DEGMINSEC
    Textfield (210,225 180x30), "%.8f", text variable: widget.field_ron_decimal, invisible if: widget.units = AxesMoveProcessWidgetUnits.DEGMINSEC
        OnMouseClick: write the text variable via VisuDialogs.Numpad
    Textfield (265,225 30x30), "%.0f", text variable: widget.field_ron_d, invisible if: widget.units <> AxesMoveProcessWidgetUnits.DEGMINSEC
        OnMouseClick: write the text variable via VisuDialogs.Numpad
    ComboBoxInteger (211,226 53x28), variable: widget.field_ron_sign, invisible if: widget.units <> AxesMoveProcessWidgetUnits.DEGMINSEC, text list: 'AxesDialogSignTextList'
    Textfield (310,225 30x30), "%.0f", text variable: widget.field_ron_m, invisible if: widget.units <> AxesMoveProcessWidgetUnits.DEGMINSEC
        OnMouseClick: write the text variable via VisuDialogs.Numpad
    Textfield (355,225 40x30), "%.1f", text variable: widget.field_ron_s, invisible if: widget.units <> AxesMoveProcessWidgetUnits.DEGMINSEC
        OnMouseClick: write the text variable via VisuDialogs.Numpad
    Label (295,225 15x30), "°", invisible if: widget.units <> AxesMoveProcessWidgetUnits.DEGMINSEC
    Label (340,225 15x30), "'", invisible if: widget.units <> AxesMoveProcessWidgetUnits.DEGMINSEC
    Label (395,225 15x30), """, invisible if: widget.units <> AxesMoveProcessWidgetUnits.DEGMINSEC
    Frame (20,30 405x25)
        shows VISU_StatusWidget(widget := widget.actualStatus)
    Rectangle (30,0 115x30), "%s", text variable: widget.title
END_VISUALIZATION

// ---- MTCS/Axes/Visu/VISU_AxesPointingModelsSetup.TcVIS
